   S707_LM_DC_2ND_CLAMP7.LS_Ret1 := FALSE;
   S707_LM_DC_2ND_CLAMP7.LS_Adv2 := FALSE;
   S707_LM_DC_2ND_CLAMP7.LS_Ret2 := FALSE;
   S707_LM_DC_2ND_CLAMP7.LS_Adv3 := FALSE;
   S707_LM_DC_2ND_CLAMP7.LS_Ret3 := FALSE;
   S707_LM_DC_2ND_CLAMP7.LS_Adv4 := FALSE;
   S707_LM_DC_2ND_CLAMP7.LS_Ret4 := FALSE;
   S707_LM_DC_2ND_CLAMP7.SOL_Adv := FALSE;
   S707_LM_DC_2ND_CLAMP7.SOL_Ret := FALSE;
   S707_LM_DC_2ND_CLAMP7.M_Ready := TRUE;
   S707_LM_DC_2ND_CLAMP7.T_CHK1 := T#4S;
   S707_LM_DC_2ND_CLAMP7.T_CHK2 := T#4S;
   S707_LM_DC_2ND_CLAMP7.PB_Lamp_CHK := FALSE;
   S707_LM_DC_2ND_CLAMP7.PB_Error_Rst := FALSE;
   S707_LM_DC_2ND_CLAMP7.M_FLICK := TRUE;
   S707_LM_DC_2ND_CLAMP7.M_Adv_Err := FALSE;
   S707_LM_DC_2ND_CLAMP7.M_Ret_Err := FALSE;
   S707_LM_DC_2ND_CLAMP7.LP_Adv := FALSE;
   S707_LM_DC_2ND_CLAMP7.LP_Ret := FALSE;
   S707_LM_DC_2ND_CLAMP7.Visu_Adv := W#16#0;
   S707_LM_DC_2ND_CLAMP7.Visu_Ret := W#16#0;
   S707_LM_DC_2ND_CLAMP7.Error_T1.IN := FALSE;
   S707_LM_DC_2ND_CLAMP7.Error_T1.PT := T#4S;
   S707_LM_DC_2ND_CLAMP7.Error_T1.Q := FALSE;
   S707_LM_DC_2ND_CLAMP7.Error_T1.ET := T#0MS;
   S707_LM_DC_2ND_CLAMP7.Error_T1.STATE := B#16#0;
   S707_LM_DC_2ND_CLAMP7.Error_T1.STIME := T#0MS;
   S707_LM_DC_2ND_CLAMP7.Error_T1.ATIME := T#0MS;
   S707_LM_DC_2ND_CLAMP7.Error_T2.IN := FALSE;
   S707_LM_DC_2ND_CLAMP7.Error_T2.PT := T#4S;
   S707_LM_DC_2ND_CLAMP7.Error_T2.Q := FALSE;
   S707_LM_DC_2ND_CLAMP7.Error_T2.ET := T#0MS;
   S707_LM_DC_2ND_CLAMP7.Error_T2.STATE := B#16#0;
   S707_LM_DC_2ND_CLAMP7.Error_T2.STIME := T#0MS;
   S707_LM_DC_2ND_CLAMP7.Error_T2.ATIME := T#0MS;
   S707_LM_DC_2ND_CLAMP7.CHK_Aux1 := FALSE;
   S707_LM_DC_2ND_CLAMP7.CHK_Aux2 := FALSE;
   S707_LM_DC_2ND_CLAMP7.Error_T1_DN := FALSE;
   S707_LM_DC_2ND_CLAMP7.Error_T2_DN := FALSE;
   S707_LM_DC_2ND_CLAMP7.Adv_Memo := TRUE;
   S707_LM_DC_2ND_CLAMP7.Visu_Adv_Arr[0] := FALSE;
   S707_LM_DC_2ND_CLAMP7.Visu_Adv_Arr[1] := FALSE;
   S707_LM_DC_2ND_CLAMP7.Visu_Adv_Arr[2] := FALSE;
   S707_LM_DC_2ND_CLAMP7.Visu_Adv_Arr[3] := FALSE;
   S707_LM_DC_2ND_CLAMP7.Visu_Adv_Arr[4] := FALSE;
   S707_LM_DC_2ND_CLAMP7.Visu_Adv_Arr[5] := FALSE;
   S707_LM_DC_2ND_CLAMP7.Visu_Adv_Arr[6] := FALSE;
   S707_LM_DC_2ND_CLAMP7.Visu_Adv_Arr[7] := FALSE;
   S707_LM_DC_2ND_CLAMP7.Visu_Adv_Arr[8] := FALSE;
   S707_LM_DC_2ND_CLAMP7.Visu_Adv_Arr[9] := FALSE;
   S707_LM_DC_2ND_CLAMP7.Visu_Adv_Arr[10] := FALSE;
   S707_LM_DC_2ND_CLAMP7.Visu_Adv_Arr[11] := FALSE;
   S707_LM_DC_2ND_CLAMP7.Visu_Adv_Arr[12] := FALSE;
   S707_LM_DC_2ND_CLAMP7.Visu_Adv_Arr[13] := FALSE;
   S707_LM_DC_2ND_CLAMP7.Visu_Adv_Arr[14] := FALSE;
   S707_LM_DC_2ND_CLAMP7.Visu_Adv_Arr[15] := FALSE;
   S707_LM_DC_2ND_CLAMP7.Visu_Ret_Arr[0] := FALSE;
   S707_LM_DC_2ND_CLAMP7.Visu_Ret_Arr[1] := FALSE;
   S707_LM_DC_2ND_CLAMP7.Visu_Ret_Arr[2] := FALSE;
   S707_LM_DC_2ND_CLAMP7.Visu_Ret_Arr[3] := FALSE;
   S707_LM_DC_2ND_CLAMP7.Visu_Ret_Arr[4] := FALSE;
   S707_LM_DC_2ND_CLAMP7.Visu_Ret_Arr[5] := FALSE;
   S707_LM_DC_2ND_CLAMP7.Visu_Ret_Arr[6] := FALSE;
   S707_LM_DC_2ND_CLAMP7.Visu_Ret_Arr[7] := FALSE;
   S707_LM_DC_2ND_CLAMP7.Visu_Ret_Arr[8] := FALSE;
   S707_LM_DC_2ND_CLAMP7.Visu_Ret_Arr[9] := FALSE;
   S707_LM_DC_2ND_CLAMP7.Visu_Ret_Arr[10] := FALSE;
   S707_LM_DC_2ND_CLAMP7.Visu_Ret_Arr[11] := FALSE;
   S707_LM_DC_2ND_CLAMP7.Visu_Ret_Arr[12] := FALSE;
   S707_LM_DC_2ND_CLAMP7.Visu_Ret_Arr[13] := FALSE;
   S707_LM_DC_2ND_CLAMP7.Visu_Ret_Arr[14] := FALSE;
   S707_LM_DC_2ND_CLAMP7.Visu_Ret_Arr[15] := FALSE;
   S707_LM_DC_2ND_CLAMP7.BLK_Move_Ret := 0;
   S707_LM_DC_2ND_CLAMP7.Enable := FALSE;
   S707_LM_DC_2ND_CLAMP7.Adv_End := FALSE;
   S707_LM_DC_2ND_CLAMP7.Ret_End := FALSE;
   S707_LM_DC_1ST_CLAMP5.Enable_Aux := FALSE;
   S707_LM_DC_1ST_CLAMP5.Adv_Amount := 1;
   S707_LM_DC_1ST_CLAMP5.Ret_Amount := 1;
   S707_LM_DC_1ST_CLAMP5.LS_Adv1 := FALSE;
   S707_LM_DC_1ST_CLAMP5.LS_Ret1 := FALSE;
   S707_LM_DC_1ST_CLAMP5.LS_Adv2 := FALSE;
   S707_LM_DC_1ST_CLAMP5.LS_Ret2 := FALSE;
   S707_LM_DC_1ST_CLAMP5.LS_Adv3 := FALSE;
   S707_LM_DC_1ST_CLAMP5.LS_Ret3 := FALSE;
   S707_LM_DC_1ST_CLAMP5.LS_Adv4 := FALSE;
   S707_LM_DC_1ST_CLAMP5.LS_Ret4 := FALSE;
   S707_LM_DC_1ST_CLAMP5.SOL_Adv := FALSE;
   S707_LM_DC_1ST_CLAMP5.SOL_Ret := FALSE;
   S707_LM_DC_1ST_CLAMP5.M_Ready := TRUE;
   S707_LM_DC_1ST_CLAMP5.T_CHK1 := T#4S;
   S707_LM_DC_1ST_CLAMP5.T_CHK2 := T#4S;
   S707_LM_DC_1ST_CLAMP5.PB_Lamp_CHK := FALSE;
   S707_LM_DC_1ST_CLAMP5.PB_Error_Rst := FALSE;
   S707_LM_DC_1ST_CLAMP5.M_FLICK := FALSE;
   S707_LM_DC_1ST_CLAMP5.M_Adv_Err := FALSE;
   S707_LM_DC_1ST_CLAMP5.M_Ret_Err := FALSE;
   S707_LM_DC_1ST_CLAMP5.LP_Adv := FALSE;
   S707_LM_DC_1ST_CLAMP5.LP_Ret := FALSE;
   S707_LM_DC_1ST_CLAMP5.Visu_Adv := W#16#0;
   S707_LM_DC_1ST_CLAMP5.Visu_Ret := W#16#0;
   S707_LM_DC_1ST_CLAMP5.Error_T1.IN := FALSE;
   S707_LM_DC_1ST_CLAMP5.Error_T1.PT := T#4S;
   S707_LM_DC_1ST_CLAMP5.Error_T1.Q := FALSE;
   S707_LM_DC_1ST_CLAMP5.Error_T1.ET := T#0MS;
   S707_LM_DC_1ST_CLAMP5.Error_T1.STATE := B#16#0;
   S707_LM_DC_1ST_CLAMP5.Error_T1.STIME := T#0MS;
   S707_LM_DC_1ST_CLAMP5.Error_T1.ATIME := T#0MS;
   S707_LM_DC_1ST_CLAMP5.Error_T2.IN := FALSE;
   S707_LM_DC_1ST_CLAMP5.Error_T2.PT := T#4S;
   S707_LM_DC_1ST_CLAMP5.Error_T2.Q := FALSE;
   S707_LM_DC_1ST_CLAMP5.Error_T2.ET := T#0MS;
   S707_LM_DC_1ST_CLAMP5.Error_T2.STATE := B#16#0;
   S707_LM_DC_1ST_CLAMP5.Error_T2.STIME := T#0MS;
   S707_LM_DC_1ST_CLAMP5.Error_T2.ATIME := T#0MS;
   S707_LM_DC_1ST_CLAMP5.CHK_Aux1 := FALSE;
   S707_LM_DC_1ST_CLAMP5.CHK_Aux2 := FALSE;
   S707_LM_DC_1ST_CLAMP5.Error_T1_DN := FALSE;
   S707_LM_DC_1ST_CLAMP5.Error_T2_DN := FALSE;
   S707_LM_DC_1ST_CLAMP5.Adv_Memo := TRUE;
   S707_LM_DC_1ST_CLAMP5.Visu_Adv_Arr[0] := FALSE;
   S707_LM_DC_1ST_CLAMP5.Visu_Adv_Arr[1] := FALSE;
   S707_LM_DC_1ST_CLAMP5.Visu_Adv_Arr[2] := FALSE;
   S707_LM_DC_1ST_CLAMP5.Visu_Adv_Arr[3] := FALSE;
   S707_LM_DC_1ST_CLAMP5.Visu_Adv_Arr[4] := FALSE;
   S707_LM_DC_1ST_CLAMP5.Visu_Adv_Arr[5] := FALSE;
   S707_LM_DC_1ST_CLAMP5.Visu_Adv_Arr[6] := FALSE;
   S707_LM_DC_1ST_CLAMP5.Visu_Adv_Arr[7] := FALSE;
   S707_LM_DC_1ST_CLAMP5.Visu_Adv_Arr[8] := FALSE;
   S707_LM_DC_1ST_CLAMP5.Visu_Adv_Arr[9] := FALSE;
   S707_LM_DC_1ST_CLAMP5.Visu_Adv_Arr[10] := FALSE;
   S707_LM_DC_1ST_CLAMP5.Visu_Adv_Arr[11] := FALSE;
   S707_LM_DC_1ST_CLAMP5.Visu_Adv_Arr[12] := FALSE;
   S707_LM_DC_1ST_CLAMP5.Visu_Adv_Arr[13] := FALSE;
   S707_LM_DC_1ST_CLAMP5.Visu_Adv_Arr[14] := FALSE;
   S707_LM_DC_1ST_CLAMP5.Visu_Adv_Arr[15] := FALSE;
   S707_LM_DC_1ST_CLAMP5.Visu_Ret_Arr[0] := FALSE;
   S707_LM_DC_1ST_CLAMP5.Visu_Ret_Arr[1] := FALSE;
   S707_LM_DC_1ST_CLAMP5.Visu_Ret_Arr[2] := FALSE;
   S707_LM_DC_1ST_CLAMP5.Visu_Ret_Arr[3] := FALSE;
   S707_LM_DC_1ST_CLAMP5.Visu_Ret_Arr[4] := FALSE;
   S707_LM_DC_1ST_CLAMP5.Visu_Ret_Arr[5] := FALSE;
   S707_LM_DC_1ST_CLAMP5.Visu_Ret_Arr[6] := FALSE;
   S707_LM_DC_1ST_CLAMP5.Visu_Ret_Arr[7] := FALSE;
   S707_LM_DC_1ST_CLAMP5.Visu_Ret_Arr[8] := FALSE;
   S707_LM_DC_1ST_CLAMP5.Visu_Ret_Arr[9] := FALSE;
   S707_LM_DC_1ST_CLAMP5.Visu_Ret_Arr[10] := FALSE;
   S707_LM_DC_1ST_CLAMP5.Visu_Ret_Arr[11] := FALSE;
   S707_LM_DC_1ST_CLAMP5.Visu_Ret_Arr[12] := FALSE;
   S707_LM_DC_1ST_CLAMP5.Visu_Ret_Arr[13] := FALSE;
   S707_LM_DC_1ST_CLAMP5.Visu_Ret_Arr[14] := FALSE;
   S707_LM_DC_1ST_CLAMP5.Visu_Ret_Arr[15] := FALSE;
   S707_LM_DC_1ST_CLAMP5.BLK_Move_Ret := 0;
   S707_LM_DC_1ST_CLAMP5.Enable := FALSE;
   S707_LM_DC_1ST_CLAMP5.Adv_End := FALSE;
   S707_LM_DC_1ST_CLAMP5.Ret_End := FALSE;
END_DATA_BLOCK

FUNCTION FC 133 : VOID
TITLE =
NAME : DAECHA
VERSION : 0.1

BEGIN
NETWORK
TITLE =
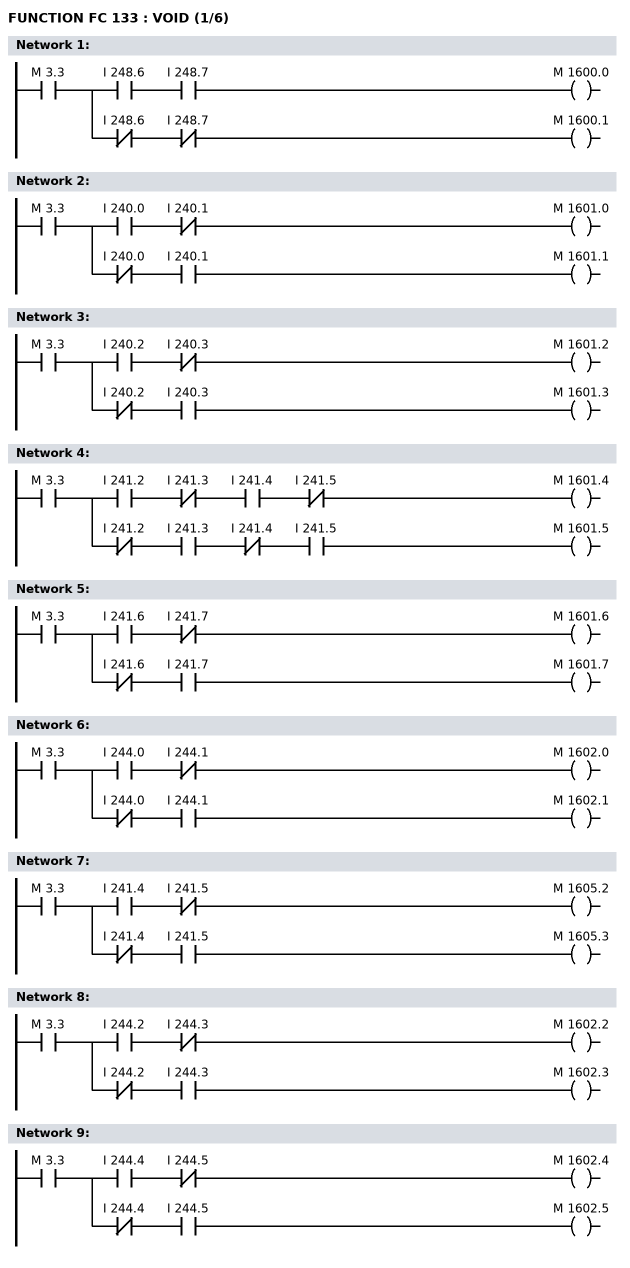

      A     M      3.3;
      =     L      0.0;
      A     L      0.0;
      A     I    248.6;
      A     I    248.7;
      =     M   1600.0;
      A     L      0.0;
      AN    I    248.6;
      AN    I    248.7;
      =     M   1600.1;
NETWORK
TITLE =

      A     M      3.3;
      =     L      0.0;
      A     L      0.0;
      A     I    240.0;
      AN    I    240.1;
      =     M   1601.0;
      A     L      0.0;
      AN    I    240.0;
      A     I    240.1;
      =     M   1601.1;
NETWORK
TITLE =

      A     M      3.3;
      =     L      0.0;
      A     L      0.0;
      A     I    240.2;
      AN    I    240.3;
      =     M   1601.2;
      A     L      0.0;
      AN    I    240.2;
      A     I    240.3;
      =     M   1601.3;
NETWORK
TITLE =

      A     M      3.3;
      =     L      0.0;
      A     L      0.0;
      A     I    241.2;
      AN    I    241.3;
      A     I    241.4;
      AN    I    241.5;
      =     M   1601.4;
      A     L      0.0;
      AN    I    241.2;
      A     I    241.3;
      AN    I    241.4;
      A     I    241.5;
      =     M   1601.5;
NETWORK
TITLE =

      A     M      3.3;
      =     L      0.0;
      A     L      0.0;
      A     I    241.6;
      AN    I    241.7;
      =     M   1601.6;
      A     L      0.0;
      AN    I    241.6;
      A     I    241.7;
      =     M   1601.7;
NETWORK
TITLE =

      A     M      3.3;
      =     L      0.0;
      A     L      0.0;
      A     I    244.0;
      AN    I    244.1;
      =     M   1602.0;
      A     L      0.0;
      AN    I    244.0;
      A     I    244.1;
      =     M   1602.1;
NETWORK
TITLE =

      A     M      3.3;
      =     L      0.0;
      A     L      0.0;
      A     I    241.4;
      AN    I    241.5;
      =     M   1605.2;
      A     L      0.0;
      AN    I    241.4;
      A     I    241.5;
      =     M   1605.3;
NETWORK
TITLE =

      A     M      3.3;
      =     L      0.0;
      A     L      0.0;
      A     I    244.2;
      AN    I    244.3;
      =     M   1602.2;
      A     L      0.0;
      AN    I    244.2;
      A     I    244.3;
      =     M   1602.3;
NETWORK
TITLE =

      A     M      3.3;
      =     L      0.0;
      A     L      0.0;
      A     I    244.4;
      AN    I    244.5;
      =     M   1602.4;
      A     L      0.0;
      AN    I    244.4;
      A     I    244.5;
      =     M   1602.5;
NETWORK
TITLE =
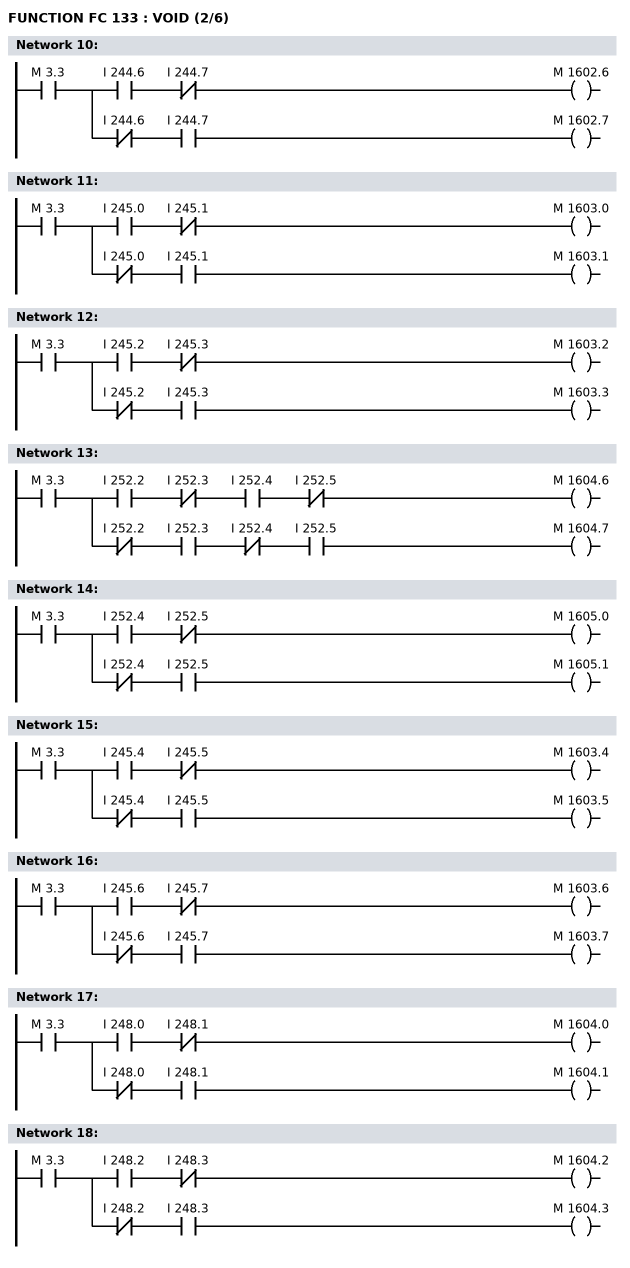

      A     M      3.3;
      =     L      0.0;
      A     L      0.0;
      A     I    244.6;
      AN    I    244.7;
      =     M   1602.6;
      A     L      0.0;
      AN    I    244.6;
      A     I    244.7;
      =     M   1602.7;
NETWORK
TITLE =

      A     M      3.3;
      =     L      0.0;
      A     L      0.0;
      A     I    245.0;
      AN    I    245.1;
      =     M   1603.0;
      A     L      0.0;
      AN    I    245.0;
      A     I    245.1;
      =     M   1603.1;
NETWORK
TITLE =

      A     M      3.3;
      =     L      0.0;
      A     L      0.0;
      A     I    245.2;
      AN    I    245.3;
      =     M   1603.2;
      A     L      0.0;
      AN    I    245.2;
      A     I    245.3;
      =     M   1603.3;
NETWORK
TITLE =

      A     M      3.3;
      =     L      0.0;
      A     L      0.0;
      A     I    252.2;
      AN    I    252.3;
      A     I    252.4;
      AN    I    252.5;
      =     M   1604.6;
      A     L      0.0;
      AN    I    252.2;
      A     I    252.3;
      AN    I    252.4;
      A     I    252.5;
      =     M   1604.7;
NETWORK
TITLE =

      A     M      3.3;
      =     L      0.0;
      A     L      0.0;
      A     I    252.4;
      AN    I    252.5;
      =     M   1605.0;
      A     L      0.0;
      AN    I    252.4;
      A     I    252.5;
      =     M   1605.1;
NETWORK
TITLE =

      A     M      3.3;
      =     L      0.0;
      A     L      0.0;
      A     I    245.4;
      AN    I    245.5;
      =     M   1603.4;
      A     L      0.0;
      AN    I    245.4;
      A     I    245.5;
      =     M   1603.5;
NETWORK
TITLE =

      A     M      3.3;
      =     L      0.0;
      A     L      0.0;
      A     I    245.6;
      AN    I    245.7;
      =     M   1603.6;
      A     L      0.0;
      AN    I    245.6;
      A     I    245.7;
      =     M   1603.7;
NETWORK
TITLE =

      A     M      3.3;
      =     L      0.0;
      A     L      0.0;
      A     I    248.0;
      AN    I    248.1;
      =     M   1604.0;
      A     L      0.0;
      AN    I    248.0;
      A     I    248.1;
      =     M   1604.1;
NETWORK
TITLE =

      A     M      3.3;
      =     L      0.0;
      A     L      0.0;
      A     I    248.2;
      AN    I    248.3;
      =     M   1604.2;
      A     L      0.0;
      AN    I    248.2;
      A     I    248.3;
      =     M   1604.3;
NETWORK
TITLE =
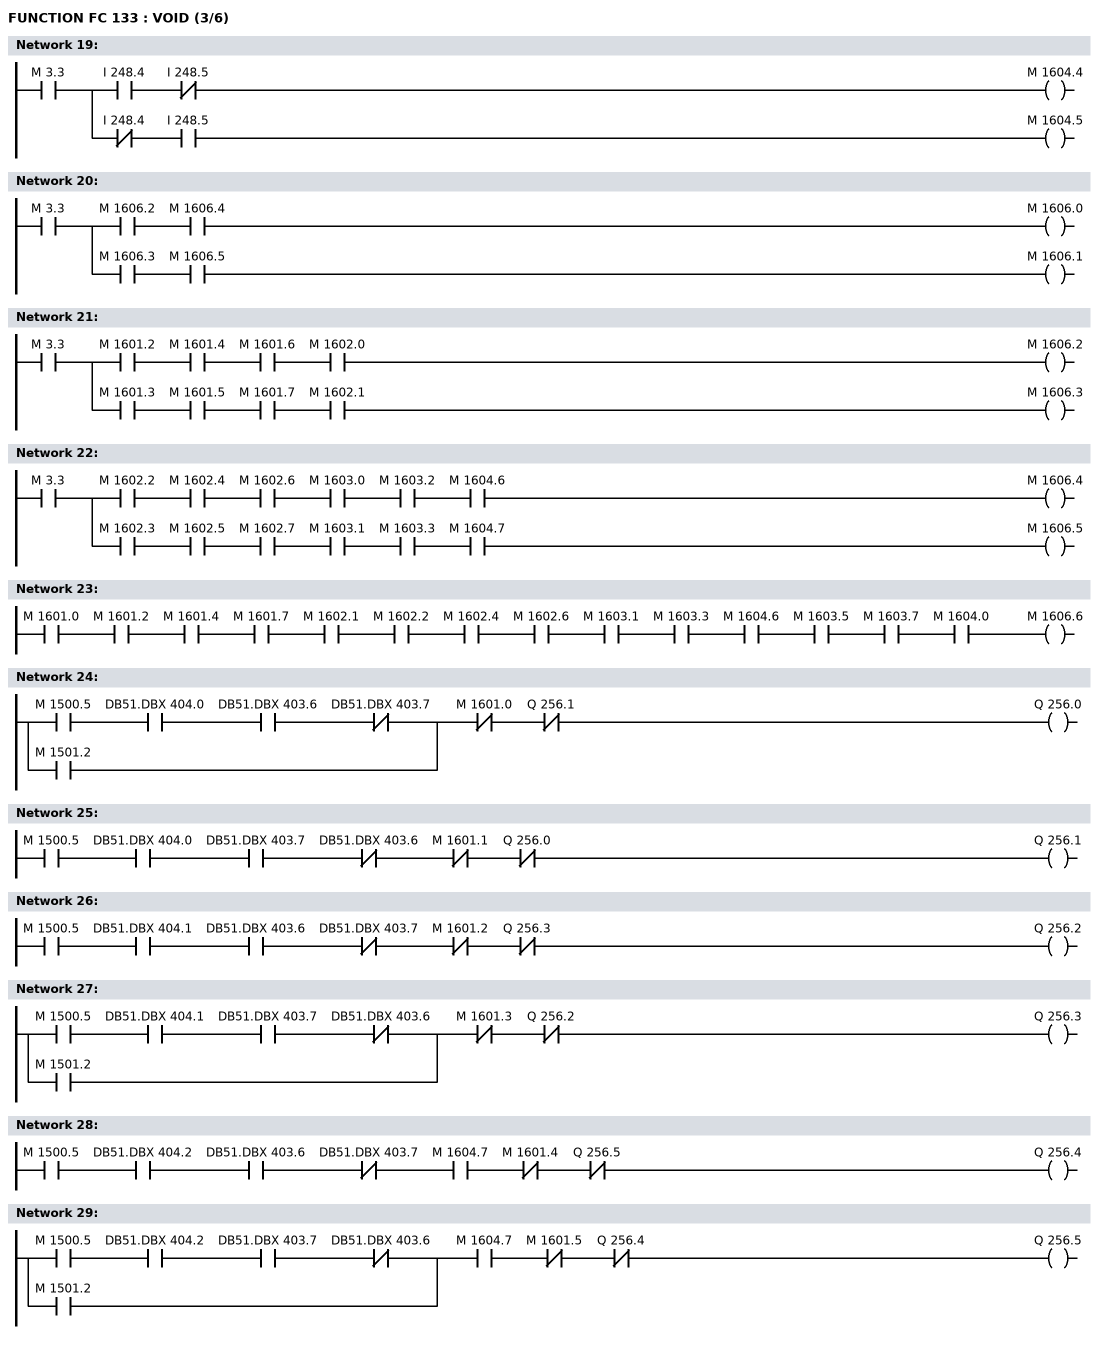

      A     M      3.3;
      =     L      0.0;
      A     L      0.0;
      A     I    248.4;
      AN    I    248.5;
      =     M   1604.4;
      A     L      0.0;
      AN    I    248.4;
      A     I    248.5;
      =     M   1604.5;
NETWORK
TITLE =

      A     M      3.3;
      =     L      0.0;
      A     L      0.0;
      A     M   1606.2;
      A     M   1606.4;
      =     M   1606.0;
      A     L      0.0;
      A     M   1606.3;
      A     M   1606.5;
      =     M   1606.1;
NETWORK
TITLE =

      A     M      3.3;
      =     L      0.0;
      A     L      0.0;
      A     M   1601.2;
      A     M   1601.4;
      A     M   1601.6;
      A     M   1602.0;
      =     M   1606.2;
      A     L      0.0;
      A     M   1601.3;
      A     M   1601.5;
      A     M   1601.7;
      A     M   1602.1;
      =     M   1606.3;
NETWORK
TITLE =

      A     M      3.3;
      =     L      0.0;
      A     L      0.0;
      A     M   1602.2;
      A     M   1602.4;
      A     M   1602.6;
      A     M   1603.0;
      A     M   1603.2;
      A     M   1604.6;
      =     M   1606.4;
      A     L      0.0;
      A     M   1602.3;
      A     M   1602.5;
      A     M   1602.7;
      A     M   1603.1;
      A     M   1603.3;
      A     M   1604.7;
      =     M   1606.5;
NETWORK
TITLE =

      A     M   1601.0;
      A     M   1601.2;
      A     M   1601.4;
      A     M   1601.7;
      A     M   1602.1;
      A     M   1602.2;
      A     M   1602.4;
      A     M   1602.6;
      A     M   1603.1;
      A     M   1603.3;
      A     M   1604.6;
      A     M   1603.5;
      A     M   1603.7;
      A     M   1604.0;
      =     M   1606.6;
NETWORK
TITLE =

      A(    ;
      A     M   1500.5;
      A     DB51.DBX  404.0;
      A     DB51.DBX  403.6;
      AN    DB51.DBX  403.7;
      O     M   1501.2;
      )     ;
      AN    M   1601.0;
      AN    Q    256.1;
      =     Q    256.0;
NETWORK
TITLE =

      A     M   1500.5;
      A     DB51.DBX  404.0;
      A     DB51.DBX  403.7;
      AN    DB51.DBX  403.6;
      AN    M   1601.1;
      AN    Q    256.0;
      =     Q    256.1;
NETWORK
TITLE =

      A     M   1500.5;
      A     DB51.DBX  404.1;
      A     DB51.DBX  403.6;
      AN    DB51.DBX  403.7;
      AN    M   1601.2;
      AN    Q    256.3;
      =     Q    256.2;
NETWORK
TITLE =

      A(    ;
      A     M   1500.5;
      A     DB51.DBX  404.1;
      A     DB51.DBX  403.7;
      AN    DB51.DBX  403.6;
      O     M   1501.2;
      )     ;
      AN    M   1601.3;
      AN    Q    256.2;
      =     Q    256.3;
NETWORK
TITLE =

      A     M   1500.5;
      A     DB51.DBX  404.2;
      A     DB51.DBX  403.6;
      AN    DB51.DBX  403.7;
      A     M   1604.7;
      AN    M   1601.4;
      AN    Q    256.5;
      =     Q    256.4;
NETWORK
TITLE =

      A(    ;
      A     M   1500.5;
      A     DB51.DBX  404.2;
      A     DB51.DBX  403.7;
      AN    DB51.DBX  403.6;
      O     M   1501.2;
      )     ;
      A     M   1604.7;
      AN    M   1601.5;
      AN    Q    256.4;
      =     Q    256.5;
NETWORK
TITLE =
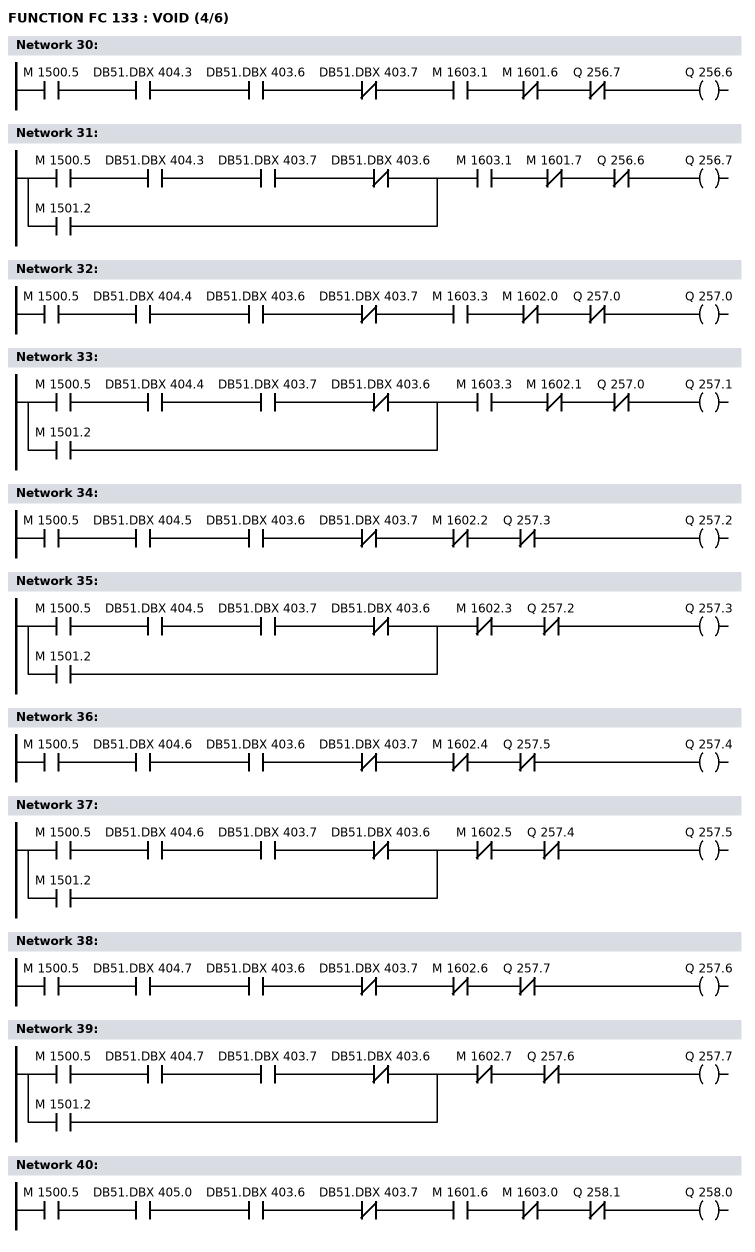

      A     M   1500.5;
      A     DB51.DBX  404.3;
      A     DB51.DBX  403.6;
      AN    DB51.DBX  403.7;
      A     M   1603.1;
      AN    M   1601.6;
      AN    Q    256.7;
      =     Q    256.6;
NETWORK
TITLE =

      A(    ;
      A     M   1500.5;
      A     DB51.DBX  404.3;
      A     DB51.DBX  403.7;
      AN    DB51.DBX  403.6;
      O     M   1501.2;
      )     ;
      A     M   1603.1;
      AN    M   1601.7;
      AN    Q    256.6;
      =     Q    256.7;
NETWORK
TITLE =

      A     M   1500.5;
      A     DB51.DBX  404.4;
      A     DB51.DBX  403.6;
      AN    DB51.DBX  403.7;
      A     M   1603.3;
      AN    M   1602.0;
      AN    Q    257.0;
      =     Q    257.0;
NETWORK
TITLE =

      A(    ;
      A     M   1500.5;
      A     DB51.DBX  404.4;
      A     DB51.DBX  403.7;
      AN    DB51.DBX  403.6;
      O     M   1501.2;
      )     ;
      A     M   1603.3;
      AN    M   1602.1;
      AN    Q    257.0;
      =     Q    257.1;
NETWORK
TITLE =

      A     M   1500.5;
      A     DB51.DBX  404.5;
      A     DB51.DBX  403.6;
      AN    DB51.DBX  403.7;
      AN    M   1602.2;
      AN    Q    257.3;
      =     Q    257.2;
NETWORK
TITLE =

      A(    ;
      A     M   1500.5;
      A     DB51.DBX  404.5;
      A     DB51.DBX  403.7;
      AN    DB51.DBX  403.6;
      O     M   1501.2;
      )     ;
      AN    M   1602.3;
      AN    Q    257.2;
      =     Q    257.3;
NETWORK
TITLE =

      A     M   1500.5;
      A     DB51.DBX  404.6;
      A     DB51.DBX  403.6;
      AN    DB51.DBX  403.7;
      AN    M   1602.4;
      AN    Q    257.5;
      =     Q    257.4;
NETWORK
TITLE =

      A(    ;
      A     M   1500.5;
      A     DB51.DBX  404.6;
      A     DB51.DBX  403.7;
      AN    DB51.DBX  403.6;
      O     M   1501.2;
      )     ;
      AN    M   1602.5;
      AN    Q    257.4;
      =     Q    257.5;
NETWORK
TITLE =

      A     M   1500.5;
      A     DB51.DBX  404.7;
      A     DB51.DBX  403.6;
      AN    DB51.DBX  403.7;
      AN    M   1602.6;
      AN    Q    257.7;
      =     Q    257.6;
NETWORK
TITLE =

      A(    ;
      A     M   1500.5;
      A     DB51.DBX  404.7;
      A     DB51.DBX  403.7;
      AN    DB51.DBX  403.6;
      O     M   1501.2;
      )     ;
      AN    M   1602.7;
      AN    Q    257.6;
      =     Q    257.7;
NETWORK
TITLE =

      A     M   1500.5;
      A     DB51.DBX  405.0;
      A     DB51.DBX  403.6;
      AN    DB51.DBX  403.7;
      A     M   1601.6;
      AN    M   1603.0;
      AN    Q    258.1;
      =     Q    258.0;
NETWORK
TITLE =
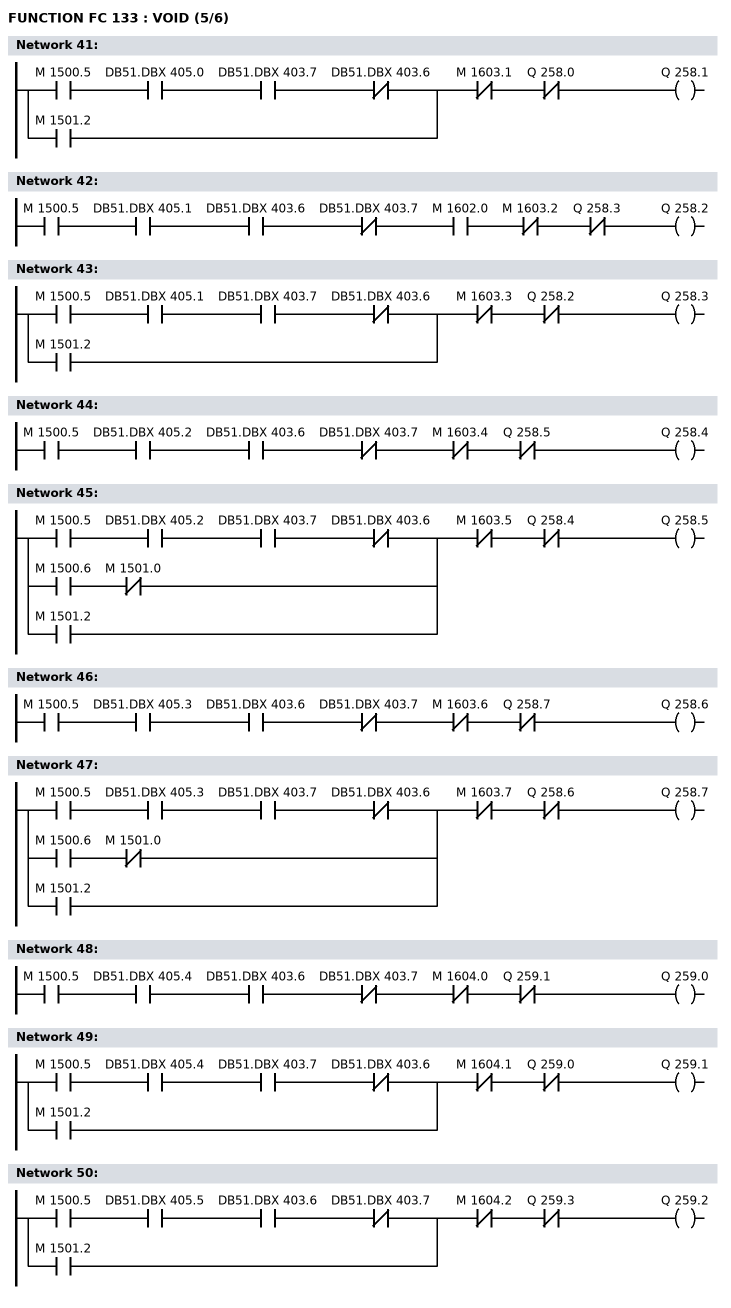

      A(    ;
      A     M   1500.5;
      A     DB51.DBX  405.0;
      A     DB51.DBX  403.7;
      AN    DB51.DBX  403.6;
      O     M   1501.2;
      )     ;
      AN    M   1603.1;
      AN    Q    258.0;
      =     Q    258.1;
NETWORK
TITLE =

      A     M   1500.5;
      A     DB51.DBX  405.1;
      A     DB51.DBX  403.6;
      AN    DB51.DBX  403.7;
      A     M   1602.0;
      AN    M   1603.2;
      AN    Q    258.3;
      =     Q    258.2;
NETWORK
TITLE =

      A(    ;
      A     M   1500.5;
      A     DB51.DBX  405.1;
      A     DB51.DBX  403.7;
      AN    DB51.DBX  403.6;
      O     M   1501.2;
      )     ;
      AN    M   1603.3;
      AN    Q    258.2;
      =     Q    258.3;
NETWORK
TITLE =

      A     M   1500.5;
      A     DB51.DBX  405.2;
      A     DB51.DBX  403.6;
      AN    DB51.DBX  403.7;
      AN    M   1603.4;
      AN    Q    258.5;
      =     Q    258.4;
NETWORK
TITLE =

      A(    ;
      A     M   1500.5;
      A     DB51.DBX  405.2;
      A     DB51.DBX  403.7;
      AN    DB51.DBX  403.6;
      O     ;
      A     M   1500.6;
      AN    M   1501.0;
      O     M   1501.2;
      )     ;
      AN    M   1603.5;
      AN    Q    258.4;
      =     Q    258.5;
NETWORK
TITLE =

      A     M   1500.5;
      A     DB51.DBX  405.3;
      A     DB51.DBX  403.6;
      AN    DB51.DBX  403.7;
      AN    M   1603.6;
      AN    Q    258.7;
      =     Q    258.6;
NETWORK
TITLE =

      A(    ;
      A     M   1500.5;
      A     DB51.DBX  405.3;
      A     DB51.DBX  403.7;
      AN    DB51.DBX  403.6;
      O     ;
      A     M   1500.6;
      AN    M   1501.0;
      O     M   1501.2;
      )     ;
      AN    M   1603.7;
      AN    Q    258.6;
      =     Q    258.7;
NETWORK
TITLE =

      A     M   1500.5;
      A     DB51.DBX  405.4;
      A     DB51.DBX  403.6;
      AN    DB51.DBX  403.7;
      AN    M   1604.0;
      AN    Q    259.1;
      =     Q    259.0;
NETWORK
TITLE =

      A(    ;
      A     M   1500.5;
      A     DB51.DBX  405.4;
      A     DB51.DBX  403.7;
      AN    DB51.DBX  403.6;
      O     M   1501.2;
      )     ;
      AN    M   1604.1;
      AN    Q    259.0;
      =     Q    259.1;
NETWORK
TITLE =

      A(    ;
      A     M   1500.5;
      A     DB51.DBX  405.5;
      A     DB51.DBX  403.6;
      AN    DB51.DBX  403.7;
      O     M   1501.2;
      )     ;
      AN    M   1604.2;
      AN    Q    259.3;
      =     Q    259.2;
NETWORK
TITLE =
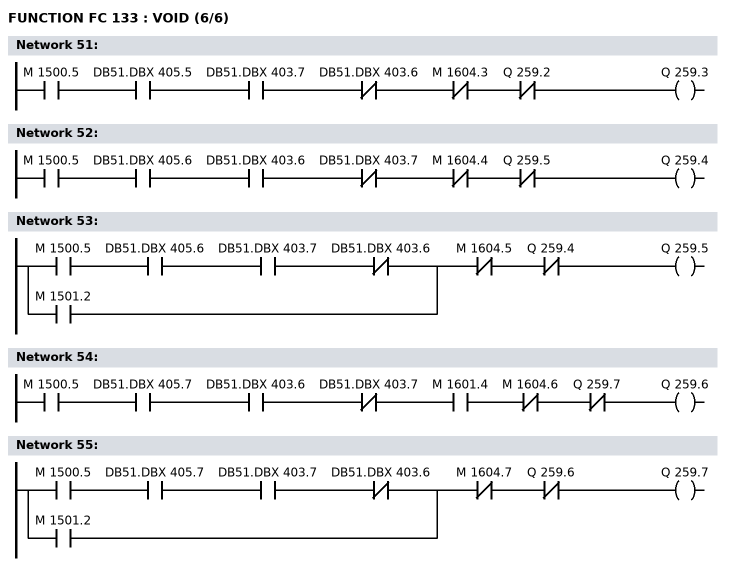

      A     M   1500.5;
      A     DB51.DBX  405.5;
      A     DB51.DBX  403.7;
      AN    DB51.DBX  403.6;
      AN    M   1604.3;
      AN    Q    259.2;
      =     Q    259.3;
NETWORK
TITLE =

      A     M   1500.5;
      A     DB51.DBX  405.6;
      A     DB51.DBX  403.6;
      AN    DB51.DBX  403.7;
      AN    M   1604.4;
      AN    Q    259.5;
      =     Q    259.4;
NETWORK
TITLE =

      A(    ;
      A     M   1500.5;
      A     DB51.DBX  405.6;
      A     DB51.DBX  403.7;
      AN    DB51.DBX  403.6;
      O     M   1501.2;
      )     ;
      AN    M   1604.5;
      AN    Q    259.4;
      =     Q    259.5;
NETWORK
TITLE =

      A     M   1500.5;
      A     DB51.DBX  405.7;
      A     DB51.DBX  403.6;
      AN    DB51.DBX  403.7;
      A     M   1601.4;
      AN    M   1604.6;
      AN    Q    259.7;
      =     Q    259.6;
NETWORK
TITLE =

      A(    ;
      A     M   1500.5;
      A     DB51.DBX  405.7;
      A     DB51.DBX  403.7;
      AN    DB51.DBX  403.6;
      O     M   1501.2;
      )     ;
      AN    M   1604.7;
      AN    Q    259.6;
      =     Q    259.7;
END_FUNCTION

FUNCTION_BLOCK FB 134
TITLE =
VERSION : 0.1


VAR
  S707_TL_DC_PIN : FB 426;
  S707_TL_DC_LATCH1 : FB 426;
  S707_TL_DC_LATCH2 : FB 426;
  S707_TL_DC_1ST_CLAMP1 : FB 426;
  S707_TL_DC_1ST_CLAMP2 : FB 426;
  S707_TL_DC_1ST_CLAMP3 : FB 426;
  S707_TL_DC_2ND_CLAMP1 : FB 426;
  S707_TL_DC_2ND_CLAMP2 : FB 426;
  S707_TL_DC_U261 : FB 426;
  S707_TL_DC_U261_CLAMP : FB 426;
  S707_TL_DC_U269 : FB 426;
  S707_TL_DC_U269_CLAMP : FB 426;
  S707_TL_DC_3RD_CLAMP : FB 426;
  S707_TL_DC_U262_1_UP_DN : FB 426;
  S707_TL_DC_U262_1 : FB 426;
  S707_TL_DC_U262_1_CLAMP : FB 426;
  S707_TL_DC_U261_2_CLAMP : FB 426;
END_VAR
BEGIN
NETWORK
TITLE =
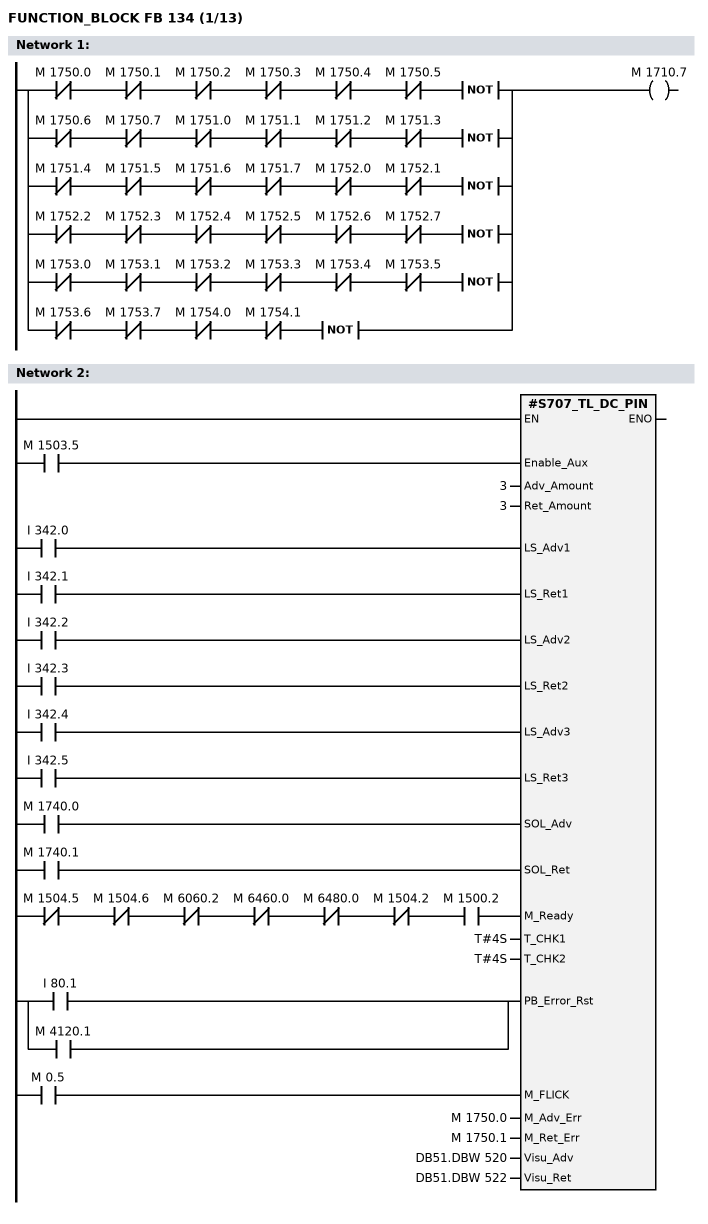

      AN    M   1750.0;
      AN    M   1750.1;
      AN    M   1750.2;
      AN    M   1750.3;
      AN    M   1750.4;
      AN    M   1750.5;
      NOT   ;
      O(    ;
      AN    M   1750.6;
      AN    M   1750.7;
      AN    M   1751.0;
      AN    M   1751.1;
      AN    M   1751.2;
      AN    M   1751.3;
      NOT   ;
      )     ;
      O(    ;
      AN    M   1751.4;
      AN    M   1751.5;
      AN    M   1751.6;
      AN    M   1751.7;
      AN    M   1752.0;
      AN    M   1752.1;
      NOT   ;
      )     ;
      O(    ;
      AN    M   1752.2;
      AN    M   1752.3;
      AN    M   1752.4;
      AN    M   1752.5;
      AN    M   1752.6;
      AN    M   1752.7;
      NOT   ;
      )     ;
      O(    ;
      AN    M   1753.0;
      AN    M   1753.1;
      AN    M   1753.2;
      AN    M   1753.3;
      AN    M   1753.4;
      AN    M   1753.5;
      NOT   ;
      )     ;
      O(    ;
      AN    M   1753.6;
      AN    M   1753.7;
      AN    M   1754.0;
      AN    M   1754.1;
      NOT   ;
      )     ;
      =     M   1710.7;
NETWORK
TITLE =

      A     M   1503.5;
      =     L      0.0;
      BLD   103;
      A     I    342.0;
      =     L      0.1;
      BLD   103;
      A     I    342.1;
      =     L      0.2;
      BLD   103;
      A     I    342.2;
      =     L      0.3;
      BLD   103;
      A     I    342.3;
      =     L      0.4;
      BLD   103;
      A     I    342.4;
      =     L      0.5;
      BLD   103;
      A     I    342.5;
      =     L      0.6;
      BLD   103;
      A     M   1740.0;
      =     L      2.1;
      BLD   103;
      A     M   1740.1;
      =     L      2.2;
      BLD   103;
      AN    M   1504.5;
      AN    M   1504.6;
      AN    M   6060.2;
      AN    M   6460.0;
      AN    M   6480.0;
      AN    M   1504.2;
      A     M   1500.2;
      =     L      2.3;
      BLD   103;
      A(    ;
      O     I     80.1;
      O     M   4120.1;
      )     ;
      =     L      2.5;
      BLD   103;
      A     M      0.5;
      =     L      2.6;
      BLD   103;
      CALL #S707_TL_DC_PIN (
           Enable_Aux               := L      0.0,
           Adv_Amount               := 3,
           Ret_Amount               := 3,
           LS_Adv1                  := L      0.1,
           LS_Ret1                  := L      0.2,
           LS_Adv2                  := L      0.3,
           LS_Ret2                  := L      0.4,
           LS_Adv3                  := L      0.5,
           LS_Ret3                  := L      0.6,
           SOL_Adv                  := L      2.1,
           SOL_Ret                  := L      2.2,
           M_Ready                  := L      2.3,
           T_CHK1                   := T#4S,
           T_CHK2                   := T#4S,
           PB_Error_Rst             := L      2.5,
           M_FLICK                  := L      2.6,
           M_Adv_Err                := M   1750.0,
           M_Ret_Err                := M   1750.1,
           Visu_Adv                 := DB51.DBW  520,
           Visu_Ret                 := DB51.DBW  522);
      NOP   0;
NETWORK
TITLE =
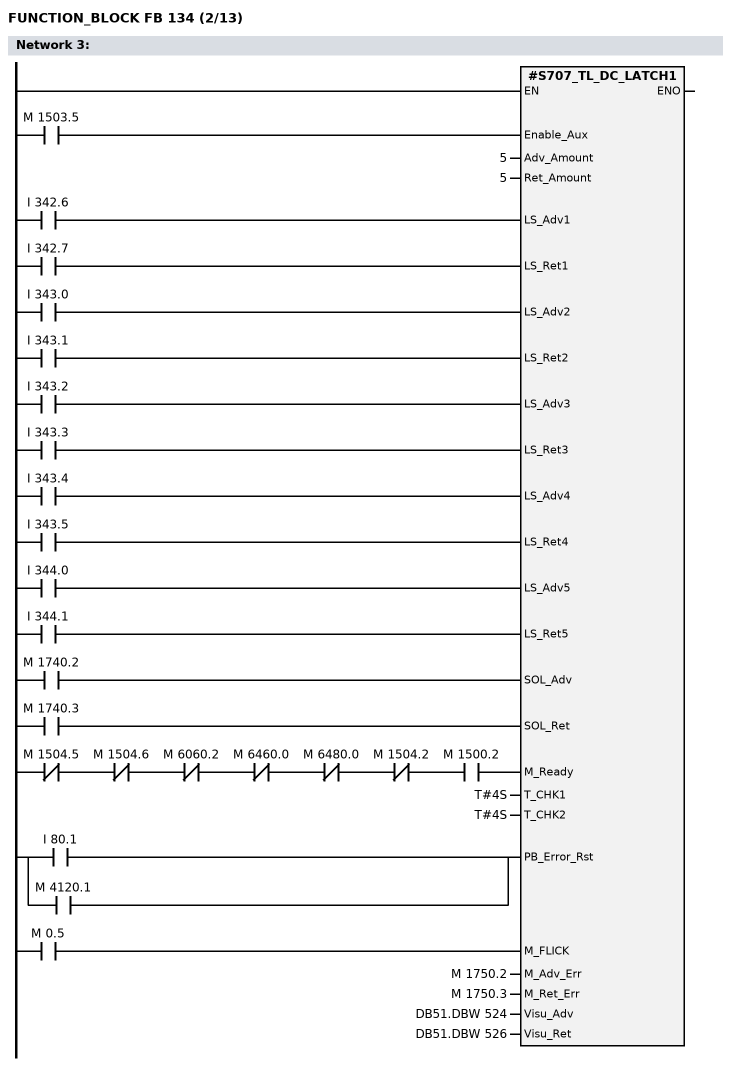

      A     M   1503.5;
      =     L      0.0;
      BLD   103;
      A     I    342.6;
      =     L      0.1;
      BLD   103;
      A     I    342.7;
      =     L      0.2;
      BLD   103;
      A     I    343.0;
      =     L      0.3;
      BLD   103;
      A     I    343.1;
      =     L      0.4;
      BLD   103;
      A     I    343.2;
      =     L      0.5;
      BLD   103;
      A     I    343.3;
      =     L      0.6;
      BLD   103;
      A     I    343.4;
      =     L      0.7;
      BLD   103;
      A     I    343.5;
      =     L      1.0;
      BLD   103;
      A     I    344.0;
      =     L      1.1;
      BLD   103;
      A     I    344.1;
      =     L      1.2;
      BLD   103;
      A     M   1740.2;
      =     L      2.1;
      BLD   103;
      A     M   1740.3;
      =     L      2.2;
      BLD   103;
      AN    M   1504.5;
      AN    M   1504.6;
      AN    M   6060.2;
      AN    M   6460.0;
      AN    M   6480.0;
      AN    M   1504.2;
      A     M   1500.2;
      =     L      2.3;
      BLD   103;
      A(    ;
      O     I     80.1;
      O     M   4120.1;
      )     ;
      =     L      2.5;
      BLD   103;
      A     M      0.5;
      =     L      2.6;
      BLD   103;
      CALL #S707_TL_DC_LATCH1 (
           Enable_Aux               := L      0.0,
           Adv_Amount               := 5,
           Ret_Amount               := 5,
           LS_Adv1                  := L      0.1,
           LS_Ret1                  := L      0.2,
           LS_Adv2                  := L      0.3,
           LS_Ret2                  := L      0.4,
           LS_Adv3                  := L      0.5,
           LS_Ret3                  := L      0.6,
           LS_Adv4                  := L      0.7,
           LS_Ret4                  := L      1.0,
           LS_Adv5                  := L      1.1,
           LS_Ret5                  := L      1.2,
           SOL_Adv                  := L      2.1,
           SOL_Ret                  := L      2.2,
           M_Ready                  := L      2.3,
           T_CHK1                   := T#4S,
           T_CHK2                   := T#4S,
           PB_Error_Rst             := L      2.5,
           M_FLICK                  := L      2.6,
           M_Adv_Err                := M   1750.2,
           M_Ret_Err                := M   1750.3,
           Visu_Adv                 := DB51.DBW  524,
           Visu_Ret                 := DB51.DBW  526);
      NOP   0;
NETWORK
TITLE =
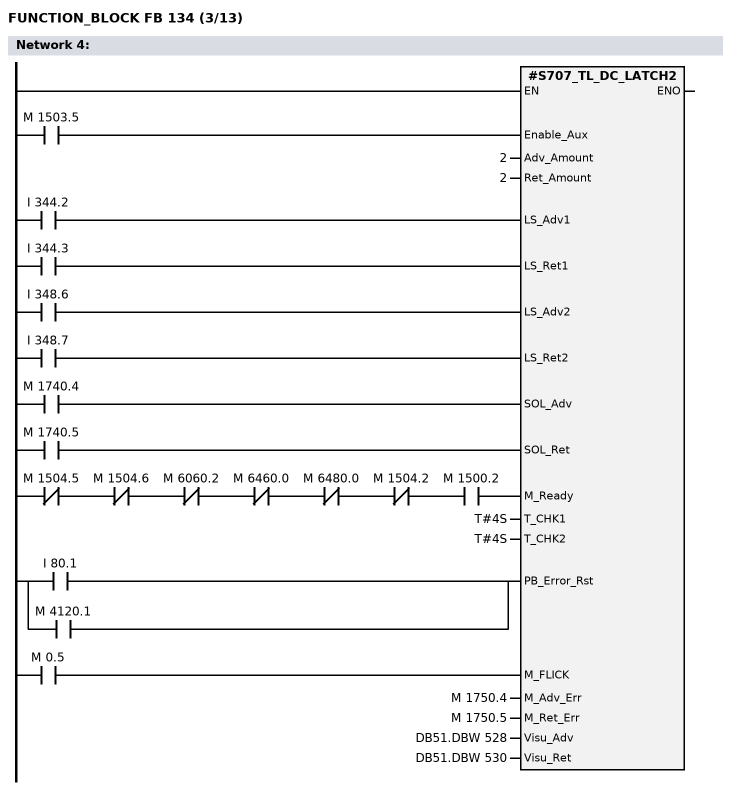

      A     M   1503.5;
      =     L      0.0;
      BLD   103;
      A     I    344.2;
      =     L      0.1;
      BLD   103;
      A     I    344.3;
      =     L      0.2;
      BLD   103;
      A     I    348.6;
      =     L      0.3;
      BLD   103;
      A     I    348.7;
      =     L      0.4;
      BLD   103;
      A     M   1740.4;
      =     L      2.1;
      BLD   103;
      A     M   1740.5;
      =     L      2.2;
      BLD   103;
      AN    M   1504.5;
      AN    M   1504.6;
      AN    M   6060.2;
      AN    M   6460.0;
      AN    M   6480.0;
      AN    M   1504.2;
      A     M   1500.2;
      =     L      2.3;
      BLD   103;
      A(    ;
      O     I     80.1;
      O     M   4120.1;
      )     ;
      =     L      2.5;
      BLD   103;
      A     M      0.5;
      =     L      2.6;
      BLD   103;
      CALL #S707_TL_DC_LATCH2 (
           Enable_Aux               := L      0.0,
           Adv_Amount               := 2,
           Ret_Amount               := 2,
           LS_Adv1                  := L      0.1,
           LS_Ret1                  := L      0.2,
           LS_Adv2                  := L      0.3,
           LS_Ret2                  := L      0.4,
           SOL_Adv                  := L      2.1,
           SOL_Ret                  := L      2.2,
           M_Ready                  := L      2.3,
           T_CHK1                   := T#4S,
           T_CHK2                   := T#4S,
           PB_Error_Rst             := L      2.5,
           M_FLICK                  := L      2.6,
           M_Adv_Err                := M   1750.4,
           M_Ret_Err                := M   1750.5,
           Visu_Adv                 := DB51.DBW  528,
           Visu_Ret                 := DB51.DBW  530);
      NOP   0;
NETWORK
TITLE =
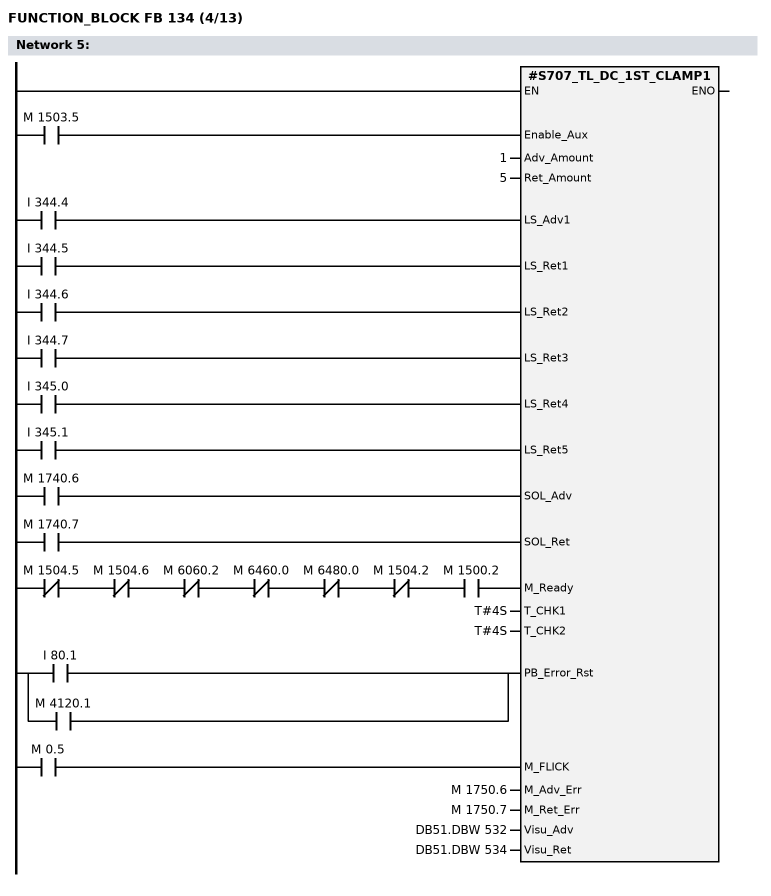

      A     M   1503.5;
      =     L      0.0;
      BLD   103;
      A     I    344.4;
      =     L      0.1;
      BLD   103;
      A     I    344.5;
      =     L      0.2;
      BLD   103;
      A     I    344.6;
      =     L      0.4;
      BLD   103;
      A     I    344.7;
      =     L      0.6;
      BLD   103;
      A     I    345.0;
      =     L      1.0;
      BLD   103;
      A     I    345.1;
      =     L      1.2;
      BLD   103;
      A     M   1740.6;
      =     L      2.1;
      BLD   103;
      A     M   1740.7;
      =     L      2.2;
      BLD   103;
      AN    M   1504.5;
      AN    M   1504.6;
      AN    M   6060.2;
      AN    M   6460.0;
      AN    M   6480.0;
      AN    M   1504.2;
      A     M   1500.2;
      =     L      2.3;
      BLD   103;
      A(    ;
      O     I     80.1;
      O     M   4120.1;
      )     ;
      =     L      2.5;
      BLD   103;
      A     M      0.5;
      =     L      2.6;
      BLD   103;
      CALL #S707_TL_DC_1ST_CLAMP1 (
           Enable_Aux               := L      0.0,
           Adv_Amount               := 1,
           Ret_Amount               := 5,
           LS_Adv1                  := L      0.1,
           LS_Ret1                  := L      0.2,
           LS_Ret2                  := L      0.4,
           LS_Ret3                  := L      0.6,
           LS_Ret4                  := L      1.0,
           LS_Ret5                  := L      1.2,
           SOL_Adv                  := L      2.1,
           SOL_Ret                  := L      2.2,
           M_Ready                  := L      2.3,
           T_CHK1                   := T#4S,
           T_CHK2                   := T#4S,
           PB_Error_Rst             := L      2.5,
           M_FLICK                  := L      2.6,
           M_Adv_Err                := M   1750.6,
           M_Ret_Err                := M   1750.7,
           Visu_Adv                 := DB51.DBW  532,
           Visu_Ret                 := DB51.DBW  534);
      NOP   0;
NETWORK
TITLE =
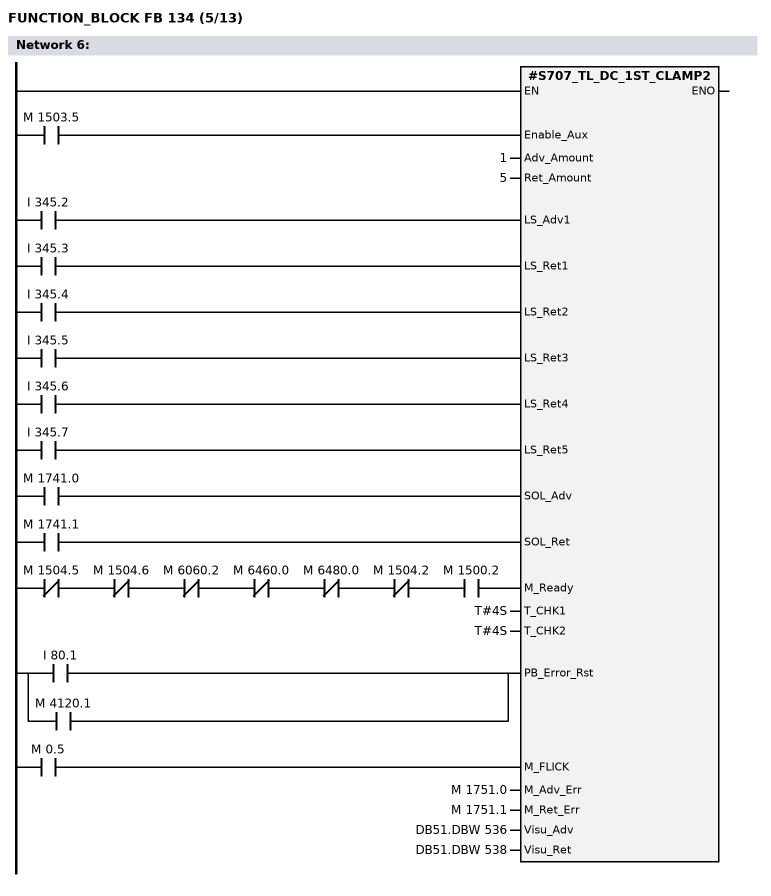

      A     M   1503.5;
      =     L      0.0;
      BLD   103;
      A     I    345.2;
      =     L      0.1;
      BLD   103;
      A     I    345.3;
      =     L      0.2;
      BLD   103;
      A     I    345.4;
      =     L      0.4;
      BLD   103;
      A     I    345.5;
      =     L      0.6;
      BLD   103;
      A     I    345.6;
      =     L      1.0;
      BLD   103;
      A     I    345.7;
      =     L      1.2;
      BLD   103;
      A     M   1741.0;
      =     L      2.1;
      BLD   103;
      A     M   1741.1;
      =     L      2.2;
      BLD   103;
      AN    M   1504.5;
      AN    M   1504.6;
      AN    M   6060.2;
      AN    M   6460.0;
      AN    M   6480.0;
      AN    M   1504.2;
      A     M   1500.2;
      =     L      2.3;
      BLD   103;
      A(    ;
      O     I     80.1;
      O     M   4120.1;
      )     ;
      =     L      2.5;
      BLD   103;
      A     M      0.5;
      =     L      2.6;
      BLD   103;
      CALL #S707_TL_DC_1ST_CLAMP2 (
           Enable_Aux               := L      0.0,
           Adv_Amount               := 1,
           Ret_Amount               := 5,
           LS_Adv1                  := L      0.1,
           LS_Ret1                  := L      0.2,
           LS_Ret2                  := L      0.4,
           LS_Ret3                  := L      0.6,
           LS_Ret4                  := L      1.0,
           LS_Ret5                  := L      1.2,
           SOL_Adv                  := L      2.1,
           SOL_Ret                  := L      2.2,
           M_Ready                  := L      2.3,
           T_CHK1                   := T#4S,
           T_CHK2                   := T#4S,
           PB_Error_Rst             := L      2.5,
           M_FLICK                  := L      2.6,
           M_Adv_Err                := M   1751.0,
           M_Ret_Err                := M   1751.1,
           Visu_Adv                 := DB51.DBW  536,
           Visu_Ret                 := DB51.DBW  538);
      NOP   0;
NETWORK
TITLE =
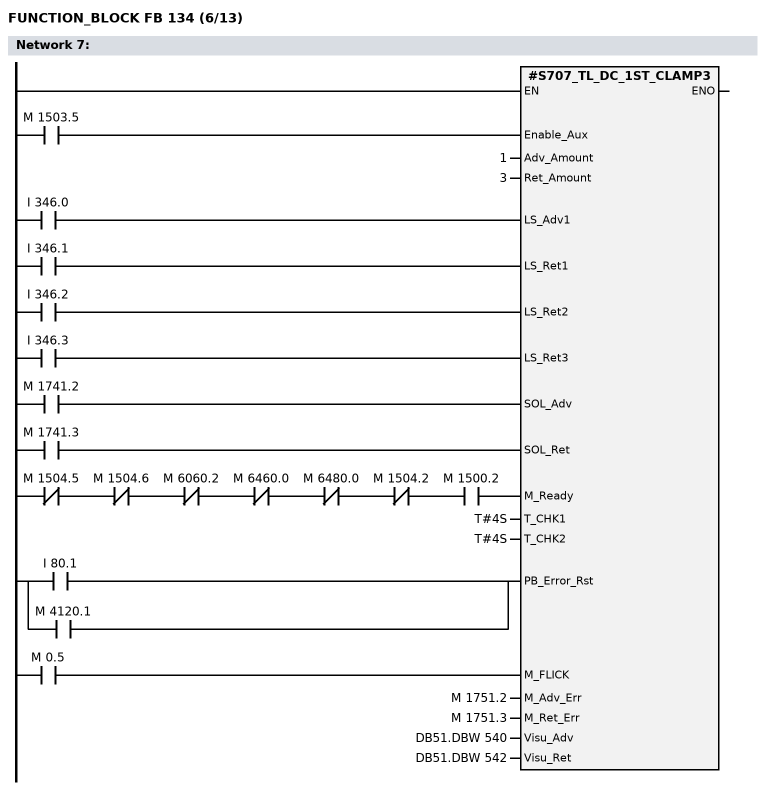

      A     M   1503.5;
      =     L      0.0;
      BLD   103;
      A     I    346.0;
      =     L      0.1;
      BLD   103;
      A     I    346.1;
      =     L      0.2;
      BLD   103;
      A     I    346.2;
      =     L      0.4;
      BLD   103;
      A     I    346.3;
      =     L      0.6;
      BLD   103;
      A     M   1741.2;
      =     L      2.1;
      BLD   103;
      A     M   1741.3;
      =     L      2.2;
      BLD   103;
      AN    M   1504.5;
      AN    M   1504.6;
      AN    M   6060.2;
      AN    M   6460.0;
      AN    M   6480.0;
      AN    M   1504.2;
      A     M   1500.2;
      =     L      2.3;
      BLD   103;
      A(    ;
      O     I     80.1;
      O     M   4120.1;
      )     ;
      =     L      2.5;
      BLD   103;
      A     M      0.5;
      =     L      2.6;
      BLD   103;
      CALL #S707_TL_DC_1ST_CLAMP3 (
           Enable_Aux               := L      0.0,
           Adv_Amount               := 1,
           Ret_Amount               := 3,
           LS_Adv1                  := L      0.1,
           LS_Ret1                  := L      0.2,
           LS_Ret2                  := L      0.4,
           LS_Ret3                  := L      0.6,
           SOL_Adv                  := L      2.1,
           SOL_Ret                  := L      2.2,
           M_Ready                  := L      2.3,
           T_CHK1                   := T#4S,
           T_CHK2                   := T#4S,
           PB_Error_Rst             := L      2.5,
           M_FLICK                  := L      2.6,
           M_Adv_Err                := M   1751.2,
           M_Ret_Err                := M   1751.3,
           Visu_Adv                 := DB51.DBW  540,
           Visu_Ret                 := DB51.DBW  542);
      NOP   0;
NETWORK
TITLE =
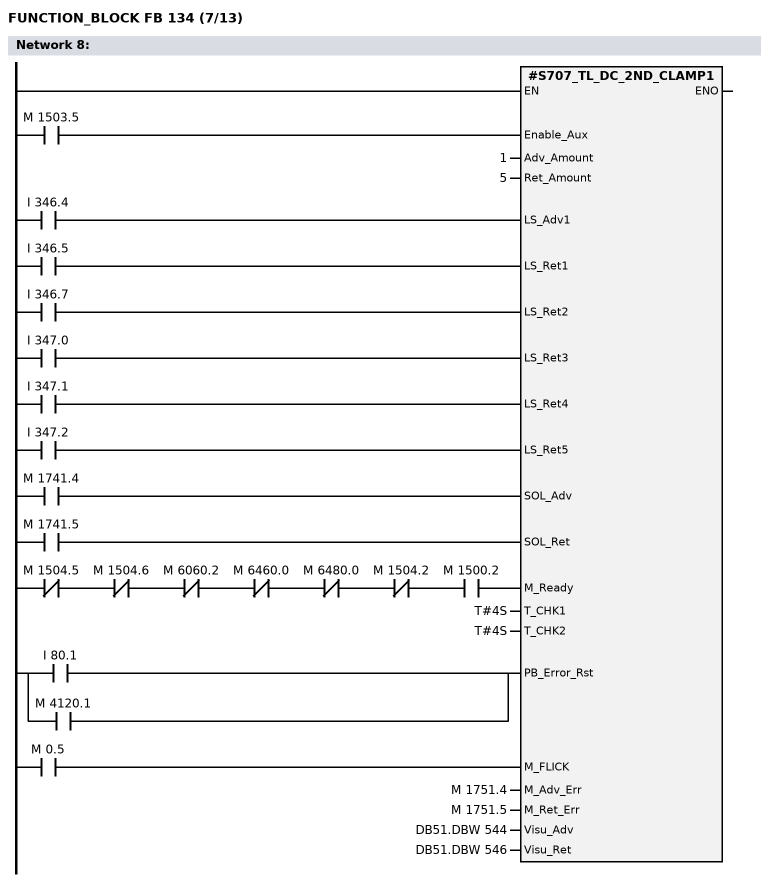

      A     M   1503.5;
      =     L      0.0;
      BLD   103;
      A     I    346.4;
      =     L      0.1;
      BLD   103;
      A     I    346.5;
      =     L      0.2;
      BLD   103;
      A     I    346.7;
      =     L      0.4;
      BLD   103;
      A     I    347.0;
      =     L      0.6;
      BLD   103;
      A     I    347.1;
      =     L      1.0;
      BLD   103;
      A     I    347.2;
      =     L      1.2;
      BLD   103;
      A     M   1741.4;
      =     L      2.1;
      BLD   103;
      A     M   1741.5;
      =     L      2.2;
      BLD   103;
      AN    M   1504.5;
      AN    M   1504.6;
      AN    M   6060.2;
      AN    M   6460.0;
      AN    M   6480.0;
      AN    M   1504.2;
      A     M   1500.2;
      =     L      2.3;
      BLD   103;
      A(    ;
      O     I     80.1;
      O     M   4120.1;
      )     ;
      =     L      2.5;
      BLD   103;
      A     M      0.5;
      =     L      2.6;
      BLD   103;
      CALL #S707_TL_DC_2ND_CLAMP1 (
           Enable_Aux               := L      0.0,
           Adv_Amount               := 1,
           Ret_Amount               := 5,
           LS_Adv1                  := L      0.1,
           LS_Ret1                  := L      0.2,
           LS_Ret2                  := L      0.4,
           LS_Ret3                  := L      0.6,
           LS_Ret4                  := L      1.0,
           LS_Ret5                  := L      1.2,
           SOL_Adv                  := L      2.1,
           SOL_Ret                  := L      2.2,
           M_Ready                  := L      2.3,
           T_CHK1                   := T#4S,
           T_CHK2                   := T#4S,
           PB_Error_Rst             := L      2.5,
           M_FLICK                  := L      2.6,
           M_Adv_Err                := M   1751.4,
           M_Ret_Err                := M   1751.5,
           Visu_Adv                 := DB51.DBW  544,
           Visu_Ret                 := DB51.DBW  546);
      NOP   0;
NETWORK
TITLE =
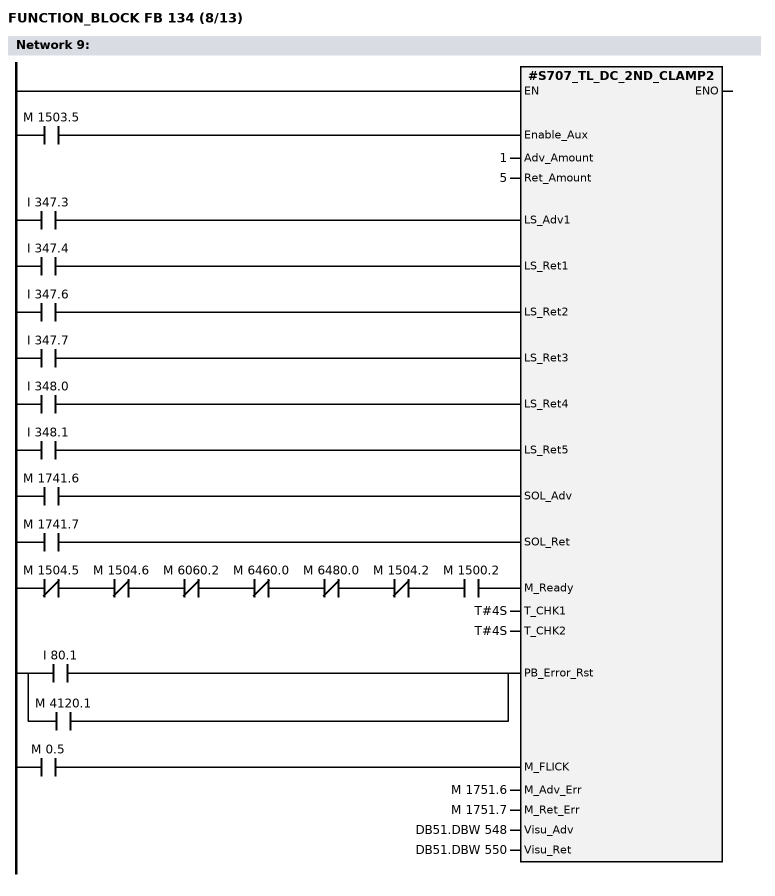

      A     M   1503.5;
      =     L      0.0;
      BLD   103;
      A     I    347.3;
      =     L      0.1;
      BLD   103;
      A     I    347.4;
      =     L      0.2;
      BLD   103;
      A     I    347.6;
      =     L      0.4;
      BLD   103;
      A     I    347.7;
      =     L      0.6;
      BLD   103;
      A     I    348.0;
      =     L      1.0;
      BLD   103;
      A     I    348.1;
      =     L      1.2;
      BLD   103;
      A     M   1741.6;
      =     L      2.1;
      BLD   103;
      A     M   1741.7;
      =     L      2.2;
      BLD   103;
      AN    M   1504.5;
      AN    M   1504.6;
      AN    M   6060.2;
      AN    M   6460.0;
      AN    M   6480.0;
      AN    M   1504.2;
      A     M   1500.2;
      =     L      2.3;
      BLD   103;
      A(    ;
      O     I     80.1;
      O     M   4120.1;
      )     ;
      =     L      2.5;
      BLD   103;
      A     M      0.5;
      =     L      2.6;
      BLD   103;
      CALL #S707_TL_DC_2ND_CLAMP2 (
           Enable_Aux               := L      0.0,
           Adv_Amount               := 1,
           Ret_Amount               := 5,
           LS_Adv1                  := L      0.1,
           LS_Ret1                  := L      0.2,
           LS_Ret2                  := L      0.4,
           LS_Ret3                  := L      0.6,
           LS_Ret4                  := L      1.0,
           LS_Ret5                  := L      1.2,
           SOL_Adv                  := L      2.1,
           SOL_Ret                  := L      2.2,
           M_Ready                  := L      2.3,
           T_CHK1                   := T#4S,
           T_CHK2                   := T#4S,
           PB_Error_Rst             := L      2.5,
           M_FLICK                  := L      2.6,
           M_Adv_Err                := M   1751.6,
           M_Ret_Err                := M   1751.7,
           Visu_Adv                 := DB51.DBW  548,
           Visu_Ret                 := DB51.DBW  550);
      NOP   0;
NETWORK
TITLE =
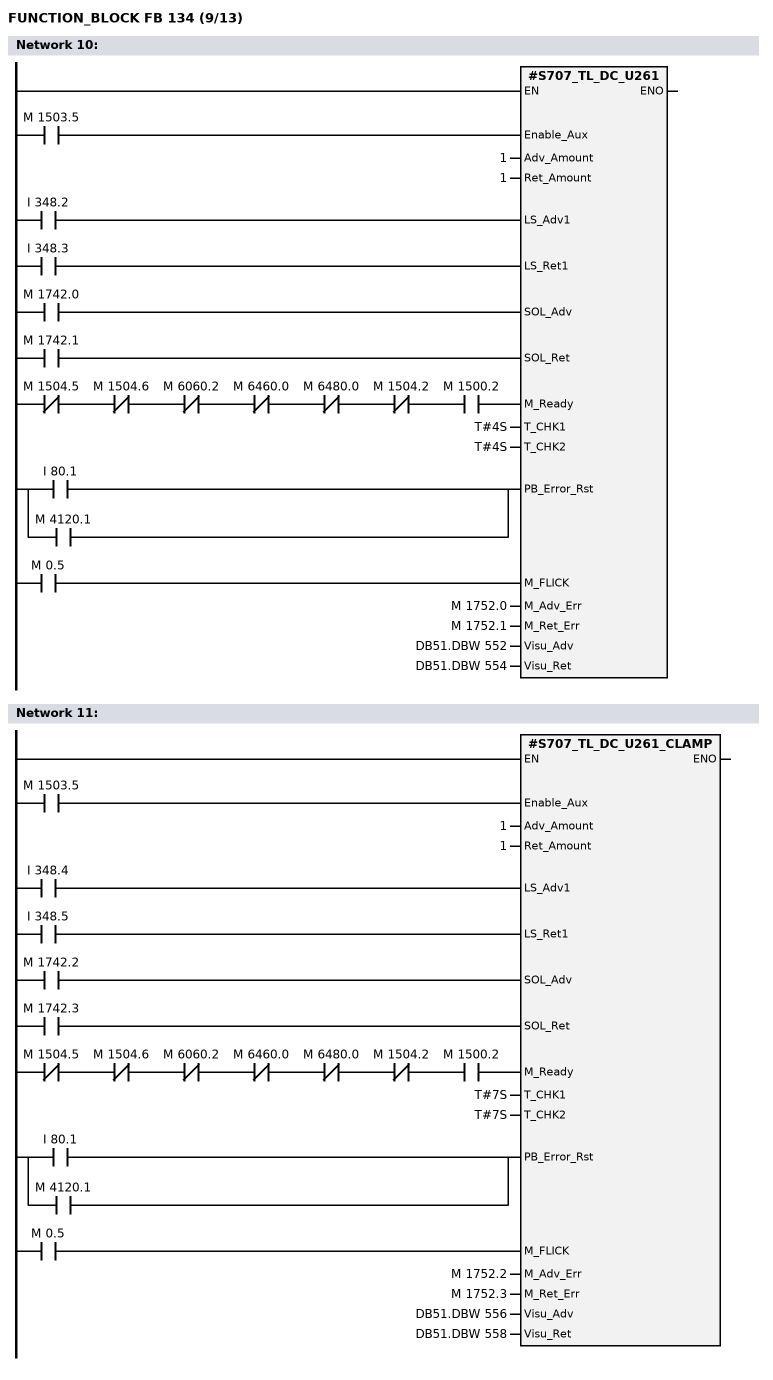

      A     M   1503.5;
      =     L      0.0;
      BLD   103;
      A     I    348.2;
      =     L      0.1;
      BLD   103;
      A     I    348.3;
      =     L      0.2;
      BLD   103;
      A     M   1742.0;
      =     L      2.1;
      BLD   103;
      A     M   1742.1;
      =     L      2.2;
      BLD   103;
      AN    M   1504.5;
      AN    M   1504.6;
      AN    M   6060.2;
      AN    M   6460.0;
      AN    M   6480.0;
      AN    M   1504.2;
      A     M   1500.2;
      =     L      2.3;
      BLD   103;
      A(    ;
      O     I     80.1;
      O     M   4120.1;
      )     ;
      =     L      2.5;
      BLD   103;
      A     M      0.5;
      =     L      2.6;
      BLD   103;
      CALL #S707_TL_DC_U261 (
           Enable_Aux               := L      0.0,
           Adv_Amount               := 1,
           Ret_Amount               := 1,
           LS_Adv1                  := L      0.1,
           LS_Ret1                  := L      0.2,
           SOL_Adv                  := L      2.1,
           SOL_Ret                  := L      2.2,
           M_Ready                  := L      2.3,
           T_CHK1                   := T#4S,
           T_CHK2                   := T#4S,
           PB_Error_Rst             := L      2.5,
           M_FLICK                  := L      2.6,
           M_Adv_Err                := M   1752.0,
           M_Ret_Err                := M   1752.1,
           Visu_Adv                 := DB51.DBW  552,
           Visu_Ret                 := DB51.DBW  554);
      NOP   0;
NETWORK
TITLE =

      A     M   1503.5;
      =     L      0.0;
      BLD   103;
      A     I    348.4;
      =     L      0.1;
      BLD   103;
      A     I    348.5;
      =     L      0.2;
      BLD   103;
      A     M   1742.2;
      =     L      2.1;
      BLD   103;
      A     M   1742.3;
      =     L      2.2;
      BLD   103;
      AN    M   1504.5;
      AN    M   1504.6;
      AN    M   6060.2;
      AN    M   6460.0;
      AN    M   6480.0;
      AN    M   1504.2;
      A     M   1500.2;
      =     L      2.3;
      BLD   103;
      A(    ;
      O     I     80.1;
      O     M   4120.1;
      )     ;
      =     L      2.5;
      BLD   103;
      A     M      0.5;
      =     L      2.6;
      BLD   103;
      CALL #S707_TL_DC_U261_CLAMP (
           Enable_Aux               := L      0.0,
           Adv_Amount               := 1,
           Ret_Amount               := 1,
           LS_Adv1                  := L      0.1,
           LS_Ret1                  := L      0.2,
           SOL_Adv                  := L      2.1,
           SOL_Ret                  := L      2.2,
           M_Ready                  := L      2.3,
           T_CHK1                   := T#7S,
           T_CHK2                   := T#7S,
           PB_Error_Rst             := L      2.5,
           M_FLICK                  := L      2.6,
           M_Adv_Err                := M   1752.2,
           M_Ret_Err                := M   1752.3,
           Visu_Adv                 := DB51.DBW  556,
           Visu_Ret                 := DB51.DBW  558);
      NOP   0;
NETWORK
TITLE =
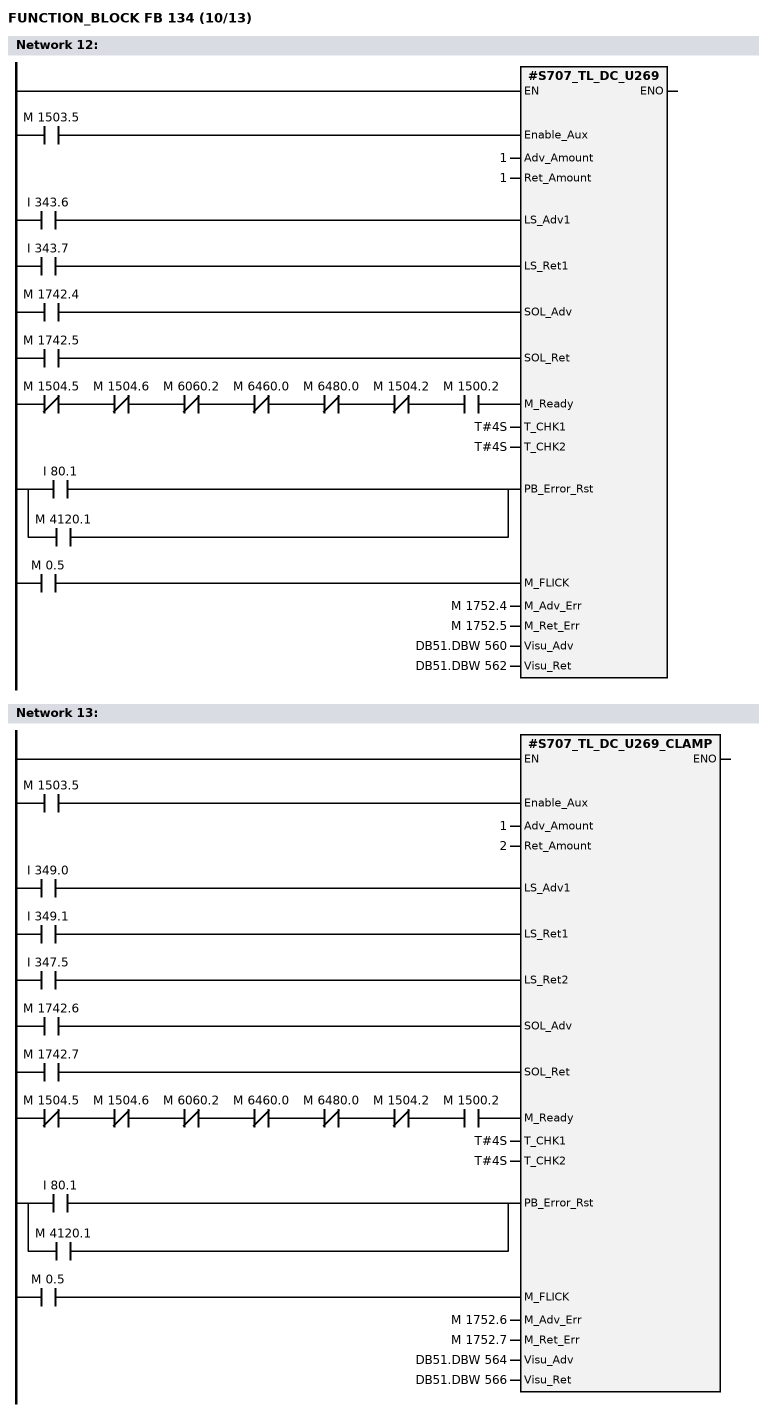

      A     M   1503.5;
      =     L      0.0;
      BLD   103;
      A     I    343.6;
      =     L      0.1;
      BLD   103;
      A     I    343.7;
      =     L      0.2;
      BLD   103;
      A     M   1742.4;
      =     L      2.1;
      BLD   103;
      A     M   1742.5;
      =     L      2.2;
      BLD   103;
      AN    M   1504.5;
      AN    M   1504.6;
      AN    M   6060.2;
      AN    M   6460.0;
      AN    M   6480.0;
      AN    M   1504.2;
      A     M   1500.2;
      =     L      2.3;
      BLD   103;
      A(    ;
      O     I     80.1;
      O     M   4120.1;
      )     ;
      =     L      2.5;
      BLD   103;
      A     M      0.5;
      =     L      2.6;
      BLD   103;
      CALL #S707_TL_DC_U269 (
           Enable_Aux               := L      0.0,
           Adv_Amount               := 1,
           Ret_Amount               := 1,
           LS_Adv1                  := L      0.1,
           LS_Ret1                  := L      0.2,
           SOL_Adv                  := L      2.1,
           SOL_Ret                  := L      2.2,
           M_Ready                  := L      2.3,
           T_CHK1                   := T#4S,
           T_CHK2                   := T#4S,
           PB_Error_Rst             := L      2.5,
           M_FLICK                  := L      2.6,
           M_Adv_Err                := M   1752.4,
           M_Ret_Err                := M   1752.5,
           Visu_Adv                 := DB51.DBW  560,
           Visu_Ret                 := DB51.DBW  562);
      NOP   0;
NETWORK
TITLE =

      A     M   1503.5;
      =     L      0.0;
      BLD   103;
      A     I    349.0;
      =     L      0.1;
      BLD   103;
      A     I    349.1;
      =     L      0.2;
      BLD   103;
      A     I    347.5;
      =     L      0.4;
      BLD   103;
      A     M   1742.6;
      =     L      2.1;
      BLD   103;
      A     M   1742.7;
      =     L      2.2;
      BLD   103;
      AN    M   1504.5;
      AN    M   1504.6;
      AN    M   6060.2;
      AN    M   6460.0;
      AN    M   6480.0;
      AN    M   1504.2;
      A     M   1500.2;
      =     L      2.3;
      BLD   103;
      A(    ;
      O     I     80.1;
      O     M   4120.1;
      )     ;
      =     L      2.5;
      BLD   103;
      A     M      0.5;
      =     L      2.6;
      BLD   103;
      CALL #S707_TL_DC_U269_CLAMP (
           Enable_Aux               := L      0.0,
           Adv_Amount               := 1,
           Ret_Amount               := 2,
           LS_Adv1                  := L      0.1,
           LS_Ret1                  := L      0.2,
           LS_Ret2                  := L      0.4,
           SOL_Adv                  := L      2.1,
           SOL_Ret                  := L      2.2,
           M_Ready                  := L      2.3,
           T_CHK1                   := T#4S,
           T_CHK2                   := T#4S,
           PB_Error_Rst             := L      2.5,
           M_FLICK                  := L      2.6,
           M_Adv_Err                := M   1752.6,
           M_Ret_Err                := M   1752.7,
           Visu_Adv                 := DB51.DBW  564,
           Visu_Ret                 := DB51.DBW  566);
      NOP   0;
NETWORK
TITLE =
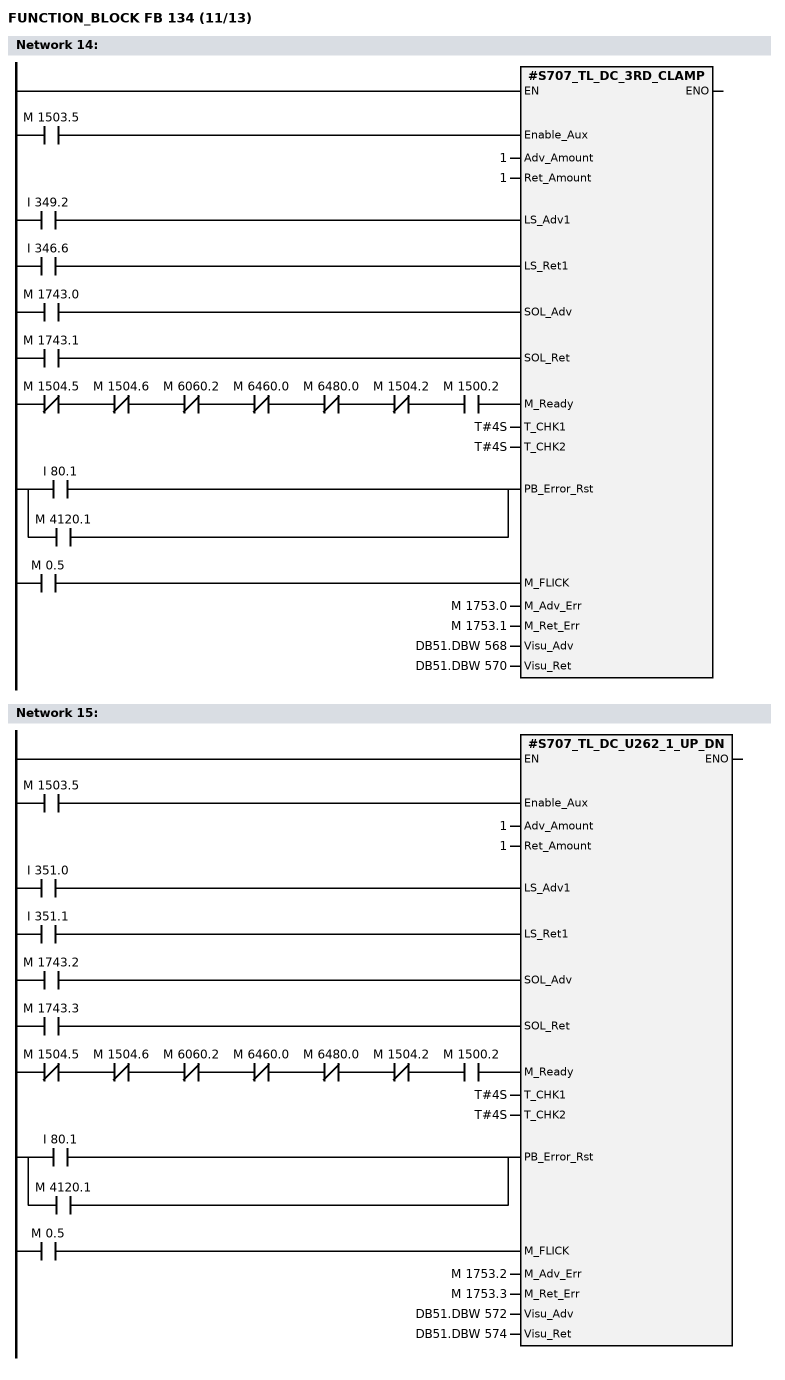

      A     M   1503.5;
      =     L      0.0;
      BLD   103;
      A     I    349.2;
      =     L      0.1;
      BLD   103;
      A     I    346.6;
      =     L      0.2;
      BLD   103;
      A     M   1743.0;
      =     L      2.1;
      BLD   103;
      A     M   1743.1;
      =     L      2.2;
      BLD   103;
      AN    M   1504.5;
      AN    M   1504.6;
      AN    M   6060.2;
      AN    M   6460.0;
      AN    M   6480.0;
      AN    M   1504.2;
      A     M   1500.2;
      =     L      2.3;
      BLD   103;
      A(    ;
      O     I     80.1;
      O     M   4120.1;
      )     ;
      =     L      2.5;
      BLD   103;
      A     M      0.5;
      =     L      2.6;
      BLD   103;
      CALL #S707_TL_DC_3RD_CLAMP (
           Enable_Aux               := L      0.0,
           Adv_Amount               := 1,
           Ret_Amount               := 1,
           LS_Adv1                  := L      0.1,
           LS_Ret1                  := L      0.2,
           SOL_Adv                  := L      2.1,
           SOL_Ret                  := L      2.2,
           M_Ready                  := L      2.3,
           T_CHK1                   := T#4S,
           T_CHK2                   := T#4S,
           PB_Error_Rst             := L      2.5,
           M_FLICK                  := L      2.6,
           M_Adv_Err                := M   1753.0,
           M_Ret_Err                := M   1753.1,
           Visu_Adv                 := DB51.DBW  568,
           Visu_Ret                 := DB51.DBW  570);
      NOP   0;
NETWORK
TITLE =

      A     M   1503.5;
      =     L      0.0;
      BLD   103;
      A     I    351.0;
      =     L      0.1;
      BLD   103;
      A     I    351.1;
      =     L      0.2;
      BLD   103;
      A     M   1743.2;
      =     L      2.1;
      BLD   103;
      A     M   1743.3;
      =     L      2.2;
      BLD   103;
      AN    M   1504.5;
      AN    M   1504.6;
      AN    M   6060.2;
      AN    M   6460.0;
      AN    M   6480.0;
      AN    M   1504.2;
      A     M   1500.2;
      =     L      2.3;
      BLD   103;
      A(    ;
      O     I     80.1;
      O     M   4120.1;
      )     ;
      =     L      2.5;
      BLD   103;
      A     M      0.5;
      =     L      2.6;
      BLD   103;
      CALL #S707_TL_DC_U262_1_UP_DN (
           Enable_Aux               := L      0.0,
           Adv_Amount               := 1,
           Ret_Amount               := 1,
           LS_Adv1                  := L      0.1,
           LS_Ret1                  := L      0.2,
           SOL_Adv                  := L      2.1,
           SOL_Ret                  := L      2.2,
           M_Ready                  := L      2.3,
           T_CHK1                   := T#4S,
           T_CHK2                   := T#4S,
           PB_Error_Rst             := L      2.5,
           M_FLICK                  := L      2.6,
           M_Adv_Err                := M   1753.2,
           M_Ret_Err                := M   1753.3,
           Visu_Adv                 := DB51.DBW  572,
           Visu_Ret                 := DB51.DBW  574);
      NOP   0;
NETWORK
TITLE =
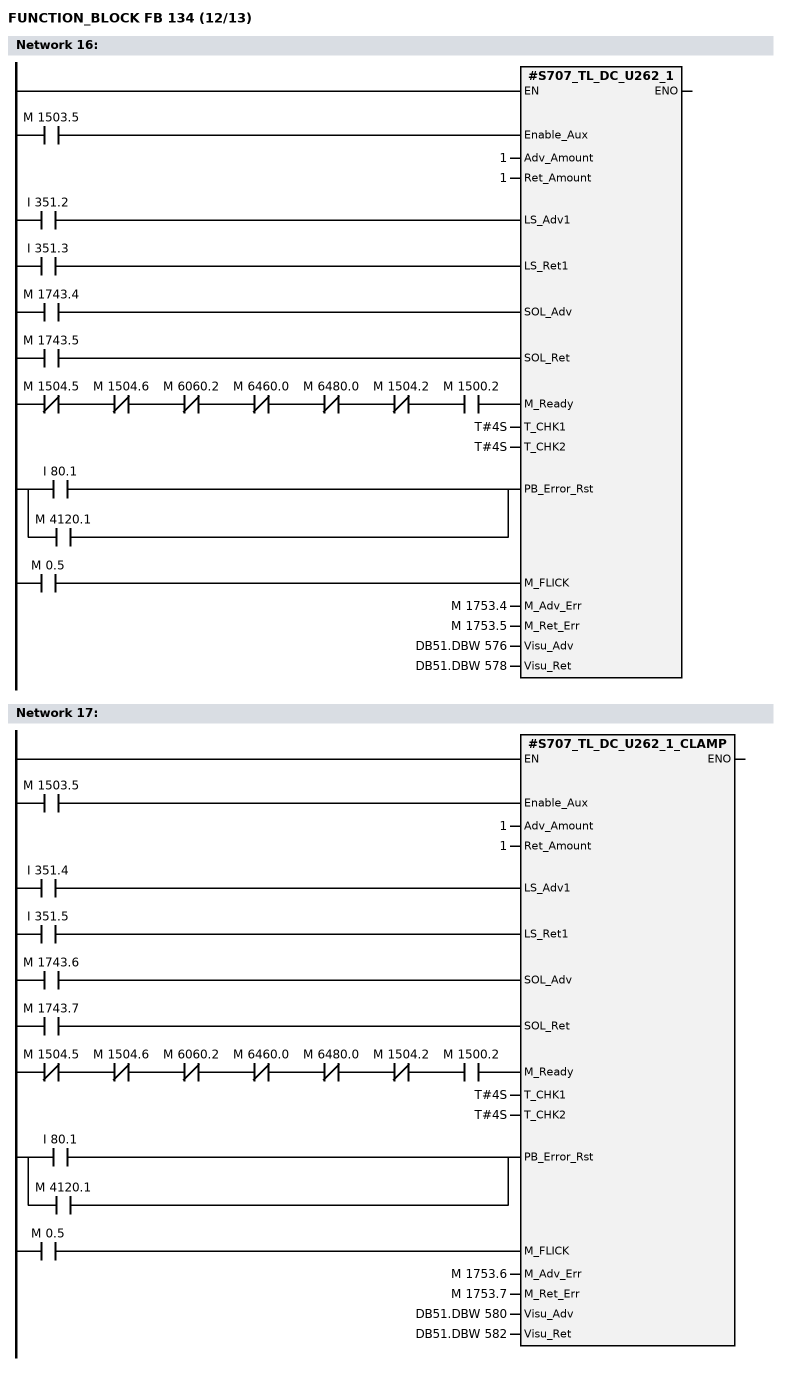

      A     M   1503.5;
      =     L      0.0;
      BLD   103;
      A     I    351.2;
      =     L      0.1;
      BLD   103;
      A     I    351.3;
      =     L      0.2;
      BLD   103;
      A     M   1743.4;
      =     L      2.1;
      BLD   103;
      A     M   1743.5;
      =     L      2.2;
      BLD   103;
      AN    M   1504.5;
      AN    M   1504.6;
      AN    M   6060.2;
      AN    M   6460.0;
      AN    M   6480.0;
      AN    M   1504.2;
      A     M   1500.2;
      =     L      2.3;
      BLD   103;
      A(    ;
      O     I     80.1;
      O     M   4120.1;
      )     ;
      =     L      2.5;
      BLD   103;
      A     M      0.5;
      =     L      2.6;
      BLD   103;
      CALL #S707_TL_DC_U262_1 (
           Enable_Aux               := L      0.0,
           Adv_Amount               := 1,
           Ret_Amount               := 1,
           LS_Adv1                  := L      0.1,
           LS_Ret1                  := L      0.2,
           SOL_Adv                  := L      2.1,
           SOL_Ret                  := L      2.2,
           M_Ready                  := L      2.3,
           T_CHK1                   := T#4S,
           T_CHK2                   := T#4S,
           PB_Error_Rst             := L      2.5,
           M_FLICK                  := L      2.6,
           M_Adv_Err                := M   1753.4,
           M_Ret_Err                := M   1753.5,
           Visu_Adv                 := DB51.DBW  576,
           Visu_Ret                 := DB51.DBW  578);
      NOP   0;
NETWORK
TITLE =

      A     M   1503.5;
      =     L      0.0;
      BLD   103;
      A     I    351.4;
      =     L      0.1;
      BLD   103;
      A     I    351.5;
      =     L      0.2;
      BLD   103;
      A     M   1743.6;
      =     L      2.1;
      BLD   103;
      A     M   1743.7;
      =     L      2.2;
      BLD   103;
      AN    M   1504.5;
      AN    M   1504.6;
      AN    M   6060.2;
      AN    M   6460.0;
      AN    M   6480.0;
      AN    M   1504.2;
      A     M   1500.2;
      =     L      2.3;
      BLD   103;
      A(    ;
      O     I     80.1;
      O     M   4120.1;
      )     ;
      =     L      2.5;
      BLD   103;
      A     M      0.5;
      =     L      2.6;
      BLD   103;
      CALL #S707_TL_DC_U262_1_CLAMP (
           Enable_Aux               := L      0.0,
           Adv_Amount               := 1,
           Ret_Amount               := 1,
           LS_Adv1                  := L      0.1,
           LS_Ret1                  := L      0.2,
           SOL_Adv                  := L      2.1,
           SOL_Ret                  := L      2.2,
           M_Ready                  := L      2.3,
           T_CHK1                   := T#4S,
           T_CHK2                   := T#4S,
           PB_Error_Rst             := L      2.5,
           M_FLICK                  := L      2.6,
           M_Adv_Err                := M   1753.6,
           M_Ret_Err                := M   1753.7,
           Visu_Adv                 := DB51.DBW  580,
           Visu_Ret                 := DB51.DBW  582);
      NOP   0;
NETWORK
TITLE =
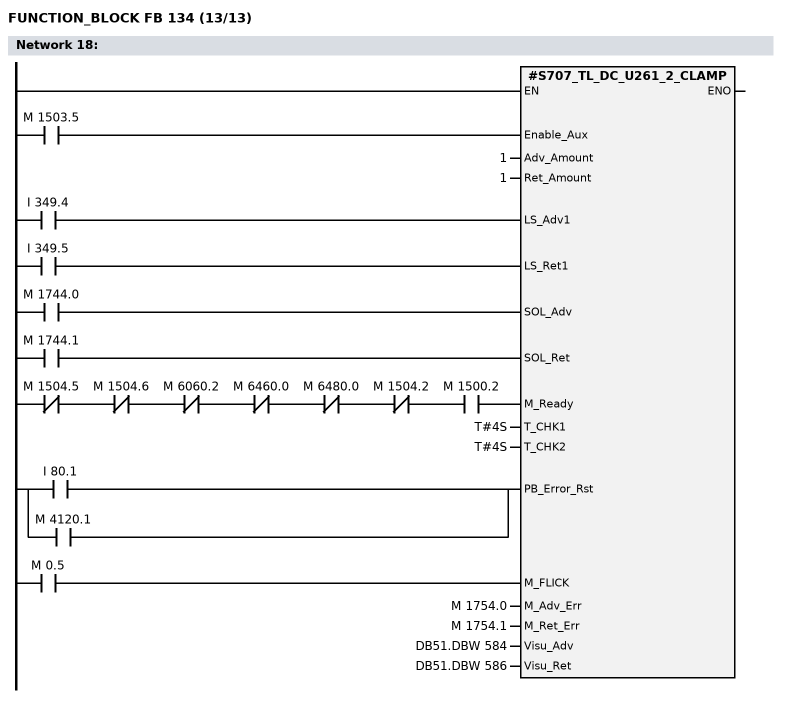

      A     M   1503.5;
      =     L      0.0;
      BLD   103;
      A     I    349.4;
      =     L      0.1;
      BLD   103;
      A     I    349.5;
      =     L      0.2;
      BLD   103;
      A     M   1744.0;
      =     L      2.1;
      BLD   103;
      A     M   1744.1;
      =     L      2.2;
      BLD   103;
      AN    M   1504.5;
      AN    M   1504.6;
      AN    M   6060.2;
      AN    M   6460.0;
      AN    M   6480.0;
      AN    M   1504.2;
      A     M   1500.2;
      =     L      2.3;
      BLD   103;
      A(    ;
      O     I     80.1;
      O     M   4120.1;
      )     ;
      =     L      2.5;
      BLD   103;
      A     M      0.5;
      =     L      2.6;
      BLD   103;
      CALL #S707_TL_DC_U261_2_CLAMP (
           Enable_Aux               := L      0.0,
           Adv_Amount               := 1,
           Ret_Amount               := 1,
           LS_Adv1                  := L      0.1,
           LS_Ret1                  := L      0.2,
           SOL_Adv                  := L      2.1,
           SOL_Ret                  := L      2.2,
           M_Ready                  := L      2.3,
           T_CHK1                   := T#4S,
           T_CHK2                   := T#4S,
           PB_Error_Rst             := L      2.5,
           M_FLICK                  := L      2.6,
           M_Adv_Err                := M   1754.0,
           M_Ret_Err                := M   1754.1,
           Visu_Adv                 := DB51.DBW  584,
           Visu_Ret                 := DB51.DBW  586);
      NOP   0;
END_FUNCTION_BLOCK

DATA_BLOCK DB 134
TITLE =
VERSION : 0.0

